LIN {X 0,Y 195.698,Z 597.397,A -85,B 0,C 180,E1 -23899.728,E2 -23899.728} C_VEL
LIN {X 0,Y 185.905,Z 599.961,A -85,B 0,C 180,E1 -23902.781,E2 -23902.781} C_VEL
LIN {X 0,Y 177.033,Z 601.325,A -85,B 0,C 180,E1 -23906.236,E2 -23906.236} C_VEL
LIN {X 0,Y 169.221,Z 601.554,A -85,B 0,C 180,E1 -23910.108,E2 -23910.108} C_VEL
LIN {X 0,Y 162.575,Z 600.655,A -85,B 0,C 180,E1 -23914.387,E2 -23914.387} C_VEL
LIN {X 0,Y 157.166,Z 598.615,A -85,B 0,C 180,E1 -23919.039,E2 -23919.039} C_VEL
LIN {X 0,Y 153.01,Z 595.413,A -85,B 0,C 180,E1 -23924.003,E2 -23924.003} C_VEL
LIN {X 0,Y 150.309,Z 590.963,A -85,B 0,C 180,E1 -23929.221,E2 -23929.221} C_VEL
LIN {X 0,Y 149.048,Z 585.18,A -85,B 0,C 180,E1 -23934.589,E2 -23934.589} C_VEL
LIN {X 0,Y 148.592,Z 577.647,A -85,B 0,C 180,E1 -23940.001,E2 -23940.001} C_VEL
LIN {X 0,Y 148.719,Z 570.72,A -85,B 0,C 180,E1 -23944.066,E2 -23944.066} C_VEL
LIN {X 0,Y 149.243,Z 562.31,A -85,B 0,C 180,E1 -23948.122,E2 -23948.122} C_VEL
LIN {X 0,Y 150.203,Z 552.102,A -85,B 0,C 180,E1 -23952.156,E2 -23952.156} C_VEL
LIN {X 0,Y 151.448,Z 540.799,A -85,B 0,C 180,E1 -23955.822,E2 -23955.822} C_VEL
LIN {X 0,Y 153.043,Z 528.174,A -85,B 0,C 180,E1 -23959.099,E2 -23959.099} C_VEL
LIN {X 0,Y 153.526,Z 523.721,A -85,B 0,C 180,E1 -23960.081,E2 -23960.081} C_VEL
LIN {X 0,Y 151.149,Z 510.343,A -85,B 0,C 180,E1 -23962.599,E2 -23962.599} C_VEL
LIN {X 0,Y 149.173,Z 497.903,A -85,B 0,C 180,E1 -23964.527,E2 -23964.527} C_VEL
LIN {X 0,Y 149.561,Z 497.851,A -85,B 0,C 180,E1 -23971.126,E2 -23971.126} C_VEL
LIN {X 0,Y 149.776,Z 497.824,A -85,B 0,C 180,E1 -23974.27,E2 -23974.27} C_VEL
LIN {X 0,Y 149.993,Z 497.8,A -85,B 0,C 180,E1 -23977.527,E2 -23977.527} C_VEL
LIN {X 0,Y 150.099,Z 497.782,A -85,B 0,C 180,E1 -23981.482,E2 -23981.482} C_VEL
LIN {X 0,Y 150.128,Z 497.783,A -85,B 0,C 180,E1 -23985.396,E2 -23985.396} C_VEL
LIN {X 0,Y 150.159,Z 497.776,A -85,B 0,C 180,E1 -23989.061,E2 -23989.061} C_VEL
LIN {X 0,Y 150.219,Z 497.772,A -85,B 0,C 180,E1 -23992.69,E2 -23992.69} C_VEL
LIN {X 0,Y 150.222,Z 497.77,A -85,B 0,C 180,E1 -23997.366,E2 -23997.366} C_VEL
LIN {X 0,Y 150.248,Z 497.769,A -85,B 0,C 180,E1 -24002.718,E2 -24002.718} C_VEL
LIN {X 0,Y 150.355,Z 497.751,A -85,B 0,C 180,E1 -24009.208,E2 -24009.208} C_VEL
LIN {X 0,Y 150.387,Z 497.752,A -85,B 0,C 180,E1 -24013.716,E2 -24013.716} C_VEL
LIN {X 0,Y 150.693,Z 497.711,A -85,B 0,C 180,E1 -24019.248,E2 -24019.248} C_VEL
LIN {X 0,Y 150.767,Z 497.706,A -85,B 0,C 180,E1 -24021.961,E2 -24021.961} C_VEL
LIN {X 0,Y 151.222,Z 497.65,A -85,B 0,C 180,E1 -24030,E2 -24030} C_VEL
LIN {X 0,Y 150.706,Z 497.714,A -85,B 0,C 180,E1 -24038.042,E2 -24038.042} C_VEL
LIN {X 0,Y 150.581,Z 497.726,A -85,B 0,C 180,E1 -24041.438,E2 -24041.438} C_VEL
LIN {X 0,Y 150.366,Z 497.755,A -85,B 0,C 180,E1 -24046.286,E2 -24046.286} C_VEL
LIN {X 0,Y 150.355,Z 497.751,A -85,B 0,C 180,E1 -24050.792,E2 -24050.792} C_VEL
LIN {X 0,Y 150.248,Z 497.769,A -85,B 0,C 180,E1 -24057.282,E2 -24057.282} C_VEL
LIN {X 0,Y 150.222,Z 497.77,A -85,B 0,C 180,E1 -24062.634,E2 -24062.634} C_VEL
LIN {X 0,Y 150.214,Z 497.773,A -85,B 0,C 180,E1 -24067.461,E2 -24067.461} C_VEL
LIN {X 0,Y 150.156,Z 497.778,A -85,B 0,C 180,E1 -24071.506,E2 -24071.506} C_VEL
LIN {X 0,Y 150.129,Z 497.784,A -85,B 0,C 180,E1 -24075.395,E2 -24075.395} C_VEL
LIN {X 0,Y 150.131,Z 497.778,A -85,B 0,C 180,E1 -24079.051,E2 -24079.051} C_VEL
LIN {X 0,Y 150.078,Z 497.79,A -85,B 0,C 180,E1 -24082.759,E2 -24082.759} C_VEL
LIN {X 0,Y 149.751,Z 497.826,A -85,B 0,C 180,E1 -24087.647,E2 -24087.647} C_VEL
LIN {X 0,Y 149.178,Z 497.898,A -85,B 0,C 180,E1 -24094.912,E2 -24094.912} C_VEL
LIN {X 0,Y 149.136,Z 497.907,A -85,B 0,C 180,E1 -24096.018,E2 -24096.018} C_VEL
LIN {X 0,Y 151.509,Z 512.126,A -85,B 0,C 180,E1 -24098.216,E2 -24098.216} C_VEL
LIN {X 0,Y 153.423,Z 522.893,A -85,B 0,C 180,E1 -24100.254,E2 -24100.254} C_VEL
LIN {X 0,Y 151.972,Z 535.306,A -85,B 0,C 180,E1 -24103.199,E2 -24103.199} C_VEL
LIN {X 0,Y 150.644,Z 546.515,A -85,B 0,C 180,E1 -24106.51,E2 -24106.51} C_VEL
LIN {X 0,Y 149.6,Z 556.661,A -85,B 0,C 180,E1 -24110.159,E2 -24110.159} C_VEL
LIN {X 0,Y 148.959,Z 565.049,A -85,B 0,C 180,E1 -24113.76,E2 -24113.76} C_VEL
LIN {X 0,Y 148.687,Z 573.127,A -85,B 0,C 180,E1 -24117.968,E2 -24117.968} C_VEL
LIN {X 0,Y 148.708,Z 580.512,A -85,B 0,C 180,E1 -24122.708,E2 -24122.708} C_VEL
LIN {X 0,Y 149.245,Z 585.686,A -85,B 0,C 180,E1 -24126.76,E2 -24126.76} C_VEL
LIN {X 0,Y 150.765,Z 591.202,A -85,B 0,C 180,E1 -24132.108,E2 -24132.108} C_VEL
LIN {X 0,Y 152.915,Z 594.451,A -85,B 0,C 180,E1 -24136.007,E2 -24136.007} C_VEL
LIN {X 0,Y 156.871,Z 597.69,A -85,B 0,C 180,E1 -24141.002,E2 -24141.002} C_VEL
LIN {X 0,Y 162.42,Z 599.76,A -85,B 0,C 180,E1 -24145.639,E2 -24145.639} C_VEL
LIN {X 0,Y 168.979,Z 600.68,A -85,B 0,C 180,E1 -24149.939,E2 -24149.939} C_VEL
LIN {X 0,Y 176.86,Z 600.442,A -85,B 0,C 180,E1 -24153.802,E2 -24153.802} C_VEL
LIN {X 0,Y 185.647,Z 599.082,A -85,B 0,C 180,E1 -24157.28,E2 -24157.28} C_VEL
LIN {X 0,Y 195.377,Z 596.535,A -85,B 0,C 180,E1 -24160.352,E2 -24160.352} C_VEL
LIN {X 0,Y 200.299,Z 594.929,A -85,B 0,C 180,E1 -24161.81,E2 -24161.81} C_VEL
LIN {X 0,Y 200.671,Z 594.93,A -85,B 0,C 180,E1 -24162.652,E2 -24162.652} C_VEL
LIN {X 0,Y 200.082,Z 595.451,A -85,B 0,C 180,E1 -24163.939,E2 -24163.939} C_VEL
LIN {X 0,Y 192.789,Z 598.957,A -85,B 0,C 180,E1 -24166.81,E2 -24166.81} C_VEL
LIN {X 0,Y 184.321,Z 602.303,A -85,B 0,C 180,E1 -24169.594,E2 -24169.594} C_VEL
LIN {X 0,Y 175.329,Z 605.126,A -85,B 0,C 180,E1 -24173.039,E2 -24173.039} C_VEL
LIN {X 0,Y 167.437,Z 606.911,A -85,B 0,C 180,E1 -24176.93,E2 -24176.93} C_VEL
LIN {X 0,Y 160.914,Z 607.677,A -85,B 0,C 180,E1 -24181.286,E2 -24181.286} C_VEL
LIN {X 0,Y 155.792,Z 607.424,A -85,B 0,C 180,E1 -24186.046,E2 -24186.046} C_VEL
LIN {X 0,Y 151.961,Z 606.089,A -85,B 0,C 180,E1 -24191.111,E2 -24191.111} C_VEL
LIN {X 0,Y 149.995,Z 603.727,A -85,B 0,C 180,E1 -24196.451,E2 -24196.451} C_VEL
LIN {X 0,Y 149.516,Z 600.172,A -85,B 0,C 180,E1 -24201.893,E2 -24201.893} C_VEL
LIN {X 0,Y 150.323,Z 595.194,A -85,B 0,C 180,E1 -24207.32,E2 -24207.32} C_VEL
LIN {X 0,Y 150.968,Z 592.887,A -85,B 0,C 180,E1 -24209.417,E2 -24209.417} C_VEL
LIN {X 0,Y 150.235,Z 596.744,A -85,B 0,C 180,E1 -24212.681,E2 -24212.681} C_VEL
LIN {X 0,Y 149.476,Z 601.603,A -85,B 0,C 180,E1 -24218.109,E2 -24218.109} C_VEL
LIN {X 0,Y 149.995,Z 605.064,A -85,B 0,C 180,E1 -24223.549,E2 -24223.549} C_VEL
LIN {X 0,Y 151.974,Z 607.36,A -85,B 0,C 180,E1 -24228.888,E2 -24228.888} C_VEL
LIN {X 0,Y 155.742,Z 608.606,A -85,B 0,C 180,E1 -24233.962,E2 -24233.962} C_VEL
LIN {X 0,Y 160.842,Z 608.816,A -85,B 0,C 180,E1 -24238.728,E2 -24238.728} C_VEL
LIN {X 0,Y 167.323,Z 608.017,A -85,B 0,C 180,E1 -24243.095,E2 -24243.095} C_VEL
LIN {X 0,Y 175.233,Z 606.214,A -85,B 0,C 180,E1 -24246.985,E2 -24246.985} C_VEL
LIN {X 0,Y 184.257,Z 603.388,A -85,B 0,C 180,E1 -24250.423,E2 -24250.423} C_VEL
LIN {X 0,Y 192.551,Z 600.121,A -85,B 0,C 180,E1 -24253.115,E2 -24253.115} C_VEL
LIN {X 0,Y 193.601,Z 599.632,A -85,B 0,C 180,E1 -24253.603,E2 -24253.603} C_VEL
LIN {X 0,Y 194.551,Z 599.052,A -85,B 0,C 180,E1 -24254.504,E2 -24254.504} C_VEL
LIN {X 0,Y 194.188,Z 598.82,A -85,B 0,C 180,E1 -24255.686,E2 -24255.686} C_VEL
LIN {X 0,Y 193.049,Z 598.915,A -85,B 0,C 180,E1 -24256.645,E2 -24256.645} C_VEL
LIN {X 0,Y 189.995,Z 599.516,A -85,B 0,C 180,E1 -24258.205,E2 -24258.205} C_VEL
LIN {X 0,Y 186.113,Z 600.31,A -85,B 0,C 180,E1 -24259.607,E2 -24259.607} C_VEL
LIN {X 0,Y 175.487,Z 601.989,A -85,B 0,C 180,E1 -24263.223,E2 -24263.223} C_VEL
LIN {X 0,Y 167.088,Z 602.317,A -85,B 0,C 180,E1 -24266.853,E2 -24266.853} C_VEL
LIN {X 0,Y 159.474,Z 601.564,A -85,B 0,C 180,E1 -24271.003,E2 -24271.003} C_VEL
LIN {X 0,Y 153.166,Z 599.679,A -85,B 0,C 180,E1 -24275.609,E2 -24275.609} C_VEL
LIN {X 0,Y 148.269,Z 596.683,A -85,B 0,C 180,E1 -24280.622,E2 -24280.622} C_VEL
LIN {X 0,Y 144.606,Z 592.483,A -85,B 0,C 180,E1 -24285.937,E2 -24285.937} C_VEL
LIN {X 0,Y 142.655,Z 587.019,A -85,B 0,C 180,E1 -24291.501,E2 -24291.501} C_VEL
LIN {X 0,Y 141.933,Z 581.951,A -85,B 0,C 180,E1 -24295.741,E2 -24295.741} C_VEL
LIN {X 0,Y 141.696,Z 574.718,A -85,B 0,C 180,E1 -24300.711,E2 -24300.711} C_VEL
LIN {X 0,Y 141.959,Z 565.75,A -85,B 0,C 180,E1 -24305.683,E2 -24305.683} C_VEL
LIN {X 0,Y 142.577,Z 557.063,A -85,B 0,C 180,E1 -24309.647,E2 -24309.647} C_VEL
LIN {X 0,Y 143.592,Z 546.908,A -85,B 0,C 180,E1 -24313.444,E2 -24313.444} C_VEL
LIN {X 0,Y 144.929,Z 535.658,A -85,B 0,C 180,E1 -24316.916,E2 -24316.916} C_VEL
LIN {X 0,Y 146.287,Z 524.84,A -85,B 0,C 180,E1 -24319.652,E2 -24319.652} C_VEL
LIN {X 0,Y 146.362,Z 523.284,A -85,B 0,C 180,E1 -24320,E2 -24320} C_VEL
LIN {X 0,Y 144.073,Z 510.803,A -85,B 0,C 180,E1 -24322.438,E2 -24322.438} C_VEL
LIN {X 0,Y 142.135,Z 498.779,A -85,B 0,C 180,E1 -24324.367,E2 -24324.367} C_VEL
LIN {X 0,Y 142.325,Z 498.755,A -85,B 0,C 180,E1 -24329.591,E2 -24329.591} C_VEL
LIN {X 0,Y 142.66,Z 498.708,A -85,B 0,C 180,E1 -24333.124,E2 -24333.124} C_VEL
LIN {X 0,Y 142.929,Z 498.682,A -85,B 0,C 180,E1 -24338.118,E2 -24338.118} C_VEL
LIN {X 0,Y 143.025,Z 498.665,A -85,B 0,C 180,E1 -24343.468,E2 -24343.468} C_VEL
LIN {X 0,Y 143.07,Z 498.662,A -85,B 0,C 180,E1 -24347.465,E2 -24347.465} C_VEL
LIN {X 0,Y 143.109,Z 498.654,A -85,B 0,C 180,E1 -24351.792,E2 -24351.792} C_VEL
LIN {X 0,Y 143.189,Z 498.646,A -85,B 0,C 180,E1 -24357.323,E2 -24357.323} C_VEL
LIN {X 0,Y 143.194,Z 498.647,A -85,B 0,C 180,E1 -24362.063,E2 -24362.063} C_VEL
LIN {X 0,Y 143.28,Z 498.633,A -85,B 0,C 180,E1 -24368.746,E2 -24368.746} C_VEL
LIN {X 0,Y 143.321,Z 498.631,A -85,B 0,C 180,E1 -24372.889,E2 -24372.889} C_VEL
LIN {X 0,Y 143.607,Z 498.594,A -85,B 0,C 180,E1 -24378.711,E2 -24378.711} C_VEL
LIN {X 0,Y 143.689,Z 498.586,A -85,B 0,C 180,E1 -24381.562,E2 -24381.562} C_VEL
LIN {X 0,Y 144.18,Z 498.527,A -85,B 0,C 180,E1 -24390,E2 -24390} C_VEL
LIN {X 0,Y 143.628,Z 498.594,A -85,B 0,C 180,E1 -24398.441,E2 -24398.441} C_VEL
LIN {X 0,Y 143.509,Z 498.606,A -85,B 0,C 180,E1 -24401.63,E2 -24401.63} C_VEL
LIN {X 0,Y 143.306,Z 498.633,A -85,B 0,C 180,E1 -24407.113,E2 -24407.113} C_VEL
LIN {X 0,Y 143.28,Z 498.633,A -85,B 0,C 180,E1 -24411.254,E2 -24411.254} C_VEL
LIN {X 0,Y 143.194,Z 498.647,A -85,B 0,C 180,E1 -24417.937,E2 -24417.937} C_VEL
LIN {X 0,Y 143.172,Z 498.649,A -85,B 0,C 180,E1 -24423.435,E2 -24423.435} C_VEL
LIN {X 0,Y 143.078,Z 498.657,A -85,B 0,C 180,E1 -24429.685,E2 -24429.685} C_VEL
LIN {X 0,Y 143.059,Z 498.665,A -85,B 0,C 180,E1 -24433.454,E2 -24433.454} C_VEL
LIN {X 0,Y 143.04,Z 498.663,A -85,B 0,C 180,E1 -24437.476,E2 -24437.476} C_VEL
LIN {X 0,Y 143.001,Z 498.673,A -85,B 0,C 180,E1 -24441.845,E2 -24441.845} C_VEL
LIN {X 0,Y 142.732,Z 498.699,A -85,B 0,C 180,E1 -24447.204,E2 -24447.204} C_VEL
LIN {X 0,Y 142.205,Z 498.77,A -85,B 0,C 180,E1 -24453.589,E2 -24453.589} C_VEL
LIN {X 0,Y 142.1,Z 498.779,A -85,B 0,C 180,E1 -24456.16,E2 -24456.16} C_VEL
LIN {X 0,Y 144.624,Z 513.6,A -85,B 0,C 180,E1 -24458.611,E2 -24458.611} C_VEL
LIN {X 0,Y 146.197,Z 522.332,A -85,B 0,C 180,E1 -24460.335,E2 -24460.335} C_VEL
LIN {X 0,Y 145.634,Z 528.278,A -85,B 0,C 180,E1 -24461.718,E2 -24461.718} C_VEL
LIN {X 0,Y 144.143,Z 540.798,A -85,B 0,C 180,E1 -24465.168,E2 -24465.168} C_VEL
LIN {X 0,Y 143.042,Z 551.16,A -85,B 0,C 180,E1 -24468.665,E2 -24468.665} C_VEL
LIN {X 0,Y 142.204,Z 561.169,A -85,B 0,C 180,E1 -24472.825,E2 -24472.825} C_VEL
LIN {X 0,Y 141.753,Z 571.068,A -85,B 0,C 180,E1 -24477.868,E2 -24477.868} C_VEL
LIN {X 0,Y 141.731,Z 577.84,A -85,B 0,C 180,E1 -24482.131,E2 -24482.131} C_VEL
LIN {X 0,Y 142.324,Z 584.32,A -85,B 0,C 180,E1 -24487.091,E2 -24487.091} C_VEL
LIN {X 0,Y 143.927,Z 590.206,A -85,B 0,C 180,E1 -24492.693,E2 -24492.693} C_VEL
LIN {X 0,Y 146.148,Z 593.742,A -85,B 0,C 180,E1 -24496.769,E2 -24496.769} C_VEL
LIN {X 0,Y 150.296,Z 597.35,A -85,B 0,C 180,E1 -24501.967,E2 -24501.967} C_VEL
LIN {X 0,Y 156.063,Z 599.826,A -85,B 0,C 180,E1 -24506.764,E2 -24506.764} C_VEL
LIN {X 0,Y 162.897,Z 601.174,A -85,B 0,C 180,E1 -24511.179,E2 -24511.179} C_VEL
LIN {X 0,Y 171.052,Z 601.383,A -85,B 0,C 180,E1 -24515.114,E2 -24515.114} C_VEL
LIN {X 0,Y 180.143,Z 600.481,A -85,B 0,C 180,E1 -24518.624,E2 -24518.624} C_VEL
LIN {X 0,Y 192.327,Z 597.879,A -85,B 0,C 180,E1 -24522.318,E2 -24522.318} C_VEL
LIN {X 0,Y 193.424,Z 597.599,A -85,B 0,C 180,E1 -24522.62,E2 -24522.62} C_VEL
LIN {X 0,Y 193.141,Z 597.833,A -85,B 0,C 180,E1 -24523.301,E2 -24523.301} C_VEL
LIN {X 0,Y 187.979,Z 599.933,A -85,B 0,C 180,E1 -24525.264,E2 -24525.264} C_VEL
LIN {X 0,Y 178.992,Z 602.901,A -85,B 0,C 180,E1 -24528.126,E2 -24528.126} C_VEL
LIN {X 0,Y 169.716,Z 605.248,A -85,B 0,C 180,E1 -24531.599,E2 -24531.599} C_VEL
LIN {X 0,Y 161.541,Z 606.599,A -85,B 0,C 180,E1 -24535.557,E2 -24535.557} C_VEL
LIN {X 0,Y 154.751,Z 606.96,A -85,B 0,C 180,E1 -24540.029,E2 -24540.029} C_VEL
LIN {X 0,Y 149.379,Z 606.337,A -85,B 0,C 180,E1 -24544.948,E2 -24544.948} C_VEL
LIN {X 0,Y 145.387,Z 604.683,A -85,B 0,C 180,E1 -24550.222,E2 -24550.222} C_VEL
LIN {X 0,Y 143.292,Z 602.031,A -85,B 0,C 180,E1 -24555.804,E2 -24555.804} C_VEL
LIN {X 0,Y 142.768,Z 598.17,A -85,B 0,C 180,E1 -24561.507,E2 -24561.507} C_VEL
LIN {X 0,Y 143.268,Z 594.348,A -85,B 0,C 180,E1 -24565.78,E2 -24565.78} C_VEL
LIN {X 0,Y 144.265,Z 590.518,A -85,B 0,C 180,E1 -24569.477,E2 -24569.477} C_VEL
LIN {X 0,Y 143.521,Z 594.455,A -85,B 0,C 180,E1 -24572.807,E2 -24572.807} C_VEL
LIN {X 0,Y 142.718,Z 599.608,A -85,B 0,C 180,E1 -24578.496,E2 -24578.496} C_VEL
LIN {X 0,Y 143.292,Z 603.359,A -85,B 0,C 180,E1 -24584.196,E2 -24584.196} C_VEL
LIN {X 0,Y 145.395,Z 605.939,A -85,B 0,C 180,E1 -24589.777,E2 -24589.777} C_VEL
LIN {X 0,Y 149.329,Z 607.531,A -85,B 0,C 180,E1 -24595.061,E2 -24595.061} C_VEL
LIN {X 0,Y 154.681,Z 608.094,A -85,B 0,C 180,E1 -24599.986,E2 -24599.986} C_VEL
LIN {X 0,Y 161.445,Z 607.693,A -85,B 0,C 180,E1 -24604.466,E2 -24604.466} C_VEL
LIN {X 0,Y 169.631,Z 606.322,A -85,B 0,C 180,E1 -24608.423,E2 -24608.423} C_VEL
LIN {X 0,Y 178.93,Z 603.954,A -85,B 0,C 180,E1 -24611.892,E2 -24611.892} C_VEL
LIN {X 0,Y 183.94,Z 602.402,A -85,B 0,C 180,E1 -24613.452,E2 -24613.452} C_VEL
LIN {X 0,Y 188.35,Z 600.741,A -85,B 0,C 180,E1 -24615.15,E2 -24615.15} C_VEL
LIN {X 0,Y 190.841,Z 599.408,A -85,B 0,C 180,E1 -24617.437,E2 -24617.437} C_VEL
LIN {X 0,Y 190.33,Z 599.383,A -85,B 0,C 180,E1 -24618.345,E2 -24618.345} C_VEL
LIN {X 0,Y 186.113,Z 600.31,A -85,B 0,C 180,E1 -24619.607,E2 -24619.607} C_VEL
LIN {X 0,Y 181.594,Z 601.229,A -85,B 0,C 180,E1 -24620.761,E2 -24620.761} C_VEL
LIN {X 0,Y 173.127,Z 602.455,A -85,B 0,C 180,E1 -24622.382,E2 -24622.382} C_VEL
LIN {X 0,Y 164.881,Z 602.98,A -85,B 0,C 180,E1 -24624.204,E2 -24624.204} C_VEL
LIN {X 0,Y 160.794,Z 602.817,A -85,B 0,C 180,E1 -24625.684,E2 -24625.684} C_VEL
LIN {X 0,Y 153.323,Z 601.682,A -85,B 0,C 180,E1 -24629.721,E2 -24629.721} C_VEL
LIN {X 0,Y 146.748,Z 599.415,A -85,B 0,C 180,E1 -24634.468,E2 -24634.468} C_VEL
LIN {X 0,Y 141.636,Z 596.05,A -85,B 0,C 180,E1 -24639.676,E2 -24639.676} C_VEL
LIN {X 0,Y 137.825,Z 591.457,A -85,B 0,C 180,E1 -24645.229,E2 -24645.229} C_VEL
LIN {X 0,Y 135.778,Z 585.648,A -85,B 0,C 180,E1 -24651.067,E2 -24651.067} C_VEL
LIN {X 0,Y 134.956,Z 579.252,A -85,B 0,C 180,E1 -24656.268,E2 -24656.268} C_VEL
LIN {X 0,Y 134.824,Z 571.474,A -85,B 0,C 180,E1 -24661.494,E2 -24661.494} C_VEL
LIN {X 0,Y 135.21,Z 562.075,A -85,B 0,C 180,E1 -24666.525,E2 -24666.525} C_VEL
LIN {X 0,Y 136.074,Z 551.25,A -85,B 0,C 180,E1 -24671.243,E2 -24671.243} C_VEL
LIN {X 0,Y 137.297,Z 540.041,A -85,B 0,C 180,E1 -24675.21,E2 -24675.21} C_VEL
LIN {X 0,Y 138.87,Z 527.241,A -85,B 0,C 180,E1 -24678.823,E2 -24678.823} C_VEL
LIN {X 0,Y 139.213,Z 524.26,A -85,B 0,C 180,E1 -24679.54,E2 -24679.54} C_VEL
LIN {X 0,Y 137.782,Z 515.546,A -85,B 0,C 180,E1 -24681.399,E2 -24681.399} C_VEL
LIN {X 0,Y 135.334,Z 501.393,A -85,B 0,C 180,E1 -24683.925,E2 -24683.925} C_VEL
LIN {X 0,Y 135.094,Z 499.655,A -85,B 0,C 180,E1 -24684.282,E2 -24684.282} C_VEL
LIN {X 0,Y 135.393,Z 499.616,A -85,B 0,C 180,E1 -24691.272,E2 -24691.272} C_VEL
LIN {X 0,Y 135.68,Z 499.582,A -85,B 0,C 180,E1 -24694.736,E2 -24694.736} C_VEL
LIN {X 0,Y 135.926,Z 499.551,A -85,B 0,C 180,E1 -24699.143,E2 -24699.143} C_VEL
LIN {X 0,Y 135.972,Z 499.544,A -85,B 0,C 180,E1 -24703.646,E2 -24703.646} C_VEL
LIN {X 0,Y 136.034,Z 499.54,A -85,B 0,C 180,E1 -24707.807,E2 -24707.807} C_VEL
LIN {X 0,Y 136.058,Z 499.532,A -85,B 0,C 180,E1 -24711.694,E2 -24711.694} C_VEL
LIN {X 0,Y 136.093,Z 499.532,A -85,B 0,C 180,E1 -24715.718,E2 -24715.718} C_VEL
LIN {X 0,Y 136.15,Z 499.526,A -85,B 0,C 180,E1 -24722.317,E2 -24722.317} C_VEL
LIN {X 0,Y 136.247,Z 499.509,A -85,B 0,C 180,E1 -24728.833,E2 -24728.833} C_VEL
LIN {X 0,Y 136.29,Z 499.505,A -85,B 0,C 180,E1 -24735.058,E2 -24735.058} C_VEL
LIN {X 0,Y 136.505,Z 499.477,A -85,B 0,C 180,E1 -24738.115,E2 -24738.115} C_VEL
LIN {X 0,Y 136.613,Z 499.467,A -85,B 0,C 180,E1 -24741.122,E2 -24741.122} C_VEL
LIN {X 0,Y 137.137,Z 499.404,A -85,B 0,C 180,E1 -24750,E2 -24750} C_VEL
LIN {X 0,Y 136.554,Z 499.474,A -85,B 0,C 180,E1 -24758.882,E2 -24758.882} C_VEL
LIN {X 0,Y 136.444,Z 499.484,A -85,B 0,C 180,E1 -24761.89,E2 -24761.89} C_VEL
LIN {X 0,Y 136.246,Z 499.514,A -85,B 0,C 180,E1 -24768.029,E2 -24768.029} C_VEL
LIN {X 0,Y 136.202,Z 499.513,A -85,B 0,C 180,E1 -24771.749,E2 -24771.749} C_VEL
LIN {X 0,Y 136.104,Z 499.528,A -85,B 0,C 180,E1 -24778.616,E2 -24778.616} C_VEL
LIN {X 0,Y 136.082,Z 499.533,A -85,B 0,C 180,E1 -24784.618,E2 -24784.618} C_VEL
LIN {X 0,Y 136.053,Z 499.532,A -85,B 0,C 180,E1 -24789.208,E2 -24789.208} C_VEL
LIN {X 0,Y 136,Z 499.545,A -85,B 0,C 180,E1 -24793.657,E2 -24793.657} C_VEL
LIN {X 0,Y 135.982,Z 499.54,A -85,B 0,C 180,E1 -24797.786,E2 -24797.786} C_VEL
LIN {X 0,Y 135.953,Z 499.55,A -85,B 0,C 180,E1 -24801.659,E2 -24801.659} C_VEL
LIN {X 0,Y 135.745,Z 499.57,A -85,B 0,C 180,E1 -24805.933,E2 -24805.933} C_VEL
LIN {X 0,Y 135.223,Z 499.64,A -85,B 0,C 180,E1 -24812.11,E2 -24812.11} C_VEL
LIN {X 0,Y 135.096,Z 499.651,A -85,B 0,C 180,E1 -24816.378,E2 -24816.378} C_VEL
LIN {X 0,Y 137.396,Z 513.137,A -85,B 0,C 180,E1 -24818.693,E2 -24818.693} C_VEL
LIN {X 0,Y 139.149,Z 523.438,A -85,B 0,C 180,E1 -24820.834,E2 -24820.834} C_VEL
LIN {X 0,Y 137.474,Z 536.858,A -85,B 0,C 180,E1 -24824.431,E2 -24824.431} C_VEL
LIN {X 0,Y 136.343,Z 547.769,A -85,B 0,C 180,E1 -24828.1,E2 -24828.1} C_VEL
LIN {X 0,Y 135.307,Z 559.508,A -85,B 0,C 180,E1 -24832.96,E2 -24832.96} C_VEL
LIN {X 0,Y 134.855,Z 568.8,A -85,B 0,C 180,E1 -24837.759,E2 -24837.759} C_VEL
LIN {X 0,Y 134.868,Z 575.931,A -85,B 0,C 180,E1 -24842.239,E2 -24842.239} C_VEL
LIN {X 0,Y 135.456,Z 582.799,A -85,B 0,C 180,E1 -24847.452,E2 -24847.452} C_VEL
LIN {X 0,Y 137.113,Z 589.071,A -85,B 0,C 180,E1 -24853.334,E2 -24853.334} C_VEL
LIN {X 0,Y 140.397,Z 593.967,A -85,B 0,C 180,E1 -24858.988,E2 -24858.988} C_VEL
LIN {X 0,Y 143.774,Z 596.869,A -85,B 0,C 180,E1 -24863.02,E2 -24863.02} C_VEL
LIN {X 0,Y 149.763,Z 599.734,A -85,B 0,C 180,E1 -24867.987,E2 -24867.987} C_VEL
LIN {X 0,Y 156.883,Z 601.486,A -85,B 0,C 180,E1 -24872.518,E2 -24872.518} C_VEL
LIN {X 0,Y 165.34,Z 602.132,A -85,B 0,C 180,E1 -24876.518,E2 -24876.518} C_VEL
LIN {X 0,Y 174.715,Z 601.69,A -85,B 0,C 180,E1 -24880.061,E2 -24880.061} C_VEL
LIN {X 0,Y 179.761,Z 601.068,A -85,B 0,C 180,E1 -24881.654,E2 -24881.654} C_VEL
LIN {X 0,Y 183.862,Z 600.524,A -85,B 0,C 180,E1 -24883.426,E2 -24883.426} C_VEL
LIN {X 0,Y 178.903,Z 602.017,A -85,B 0,C 180,E1 -24885,E2 -24885} C_VEL
LIN {X 0,Y 168.885,Z 604.384,A -85,B 0,C 180,E1 -24888.254,E2 -24888.254} C_VEL
LIN {X 0,Y 159.927,Z 605.788,A -85,B 0,C 180,E1 -24892.031,E2 -24892.031} C_VEL
LIN {X 0,Y 151.774,Z 606.22,A -85,B 0,C 180,E1 -24896.46,E2 -24896.46} C_VEL
LIN {X 0,Y 145.667,Z 605.717,A -85,B 0,C 180,E1 -24901.153,E2 -24901.153} C_VEL
LIN {X 0,Y 140.776,Z 604.247,A -85,B 0,C 180,E1 -24906.46,E2 -24906.46} C_VEL
LIN {X 0,Y 137.516,Z 601.771,A -85,B 0,C 180,E1 -24912.143,E2 -24912.143} C_VEL
LIN {X 0,Y 136.069,Z 597.67,A -85,B 0,C 180,E1 -24918.916,E2 -24918.916} C_VEL
LIN {X 0,Y 136.36,Z 593.416,A -85,B 0,C 180,E1 -24924.083,E2 -24924.083} C_VEL
LIN {X 0,Y 137.676,Z 587.892,A -85,B 0,C 180,E1 -24929.452,E2 -24929.452} C_VEL
LIN {X 0,Y 136.52,Z 593.578,A -85,B 0,C 180,E1 -24934.429,E2 -24934.429} C_VEL
LIN {X 0,Y 136.057,Z 599.045,A -85,B 0,C 180,E1 -24941.057,E2 -24941.057} C_VEL
LIN {X 0,Y 136.63,Z 601.524,A -85,B 0,C 180,E1 -24944.903,E2 -24944.903} C_VEL
LIN {X 0,Y 138.871,Z 604.406,A -85,B 0,C 180,E1 -24950.748,E2 -24950.748} C_VEL
LIN {X 0,Y 143.001,Z 606.304,A -85,B 0,C 180,E1 -24956.252,E2 -24956.252} C_VEL
LIN {X 0,Y 148.6,Z 607.22,A -85,B 0,C 180,E1 -24961.349,E2 -24961.349} C_VEL
LIN {X 0,Y 155.662,Z 607.204,A -85,B 0,C 180,E1 -24965.94,E2 -24965.94} C_VEL
LIN {X 0,Y 164.134,Z 606.261,A -85,B 0,C 180,E1 -24969.962,E2 -24969.962} C_VEL
LIN {X 0,Y 173.716,Z 604.359,A -85,B 0,C 180,E1 -24973.454,E2 -24973.454} C_VEL
LIN {X 0,Y 178.874,Z 603.043,A -85,B 0,C 180,E1 -24975.01,E2 -24975.01} C_VEL
LIN {X 0,Y 182.905,Z 601.689,A -85,B 0,C 180,E1 -24976.892,E2 -24976.892} C_VEL
LIN {X 0,Y 180.033,Z 601.984,A -85,B 0,C 180,E1 -24978.423,E2 -24978.423} C_VEL
LIN {X 0,Y 169.91,Z 602.975,A -85,B 0,C 180,E1 -24981.804,E2 -24981.804} C_VEL
LIN {X 0,Y 160.794,Z 602.817,A -85,B 0,C 180,E1 -24985.684,E2 -24985.684} C_VEL
LIN {X 0,Y 156.842,Z 602.474,A -85,B 0,C 180,E1 -24987.265,E2 -24987.265} C_VEL
LIN {X 0,Y 149.307,Z 601.394,A -85,B 0,C 180,E1 -24989.651,E2 -24989.651} C_VEL
LIN {X 0,Y 142.286,Z 599.63,A -85,B 0,C 180,E1 -24992.298,E2 -24992.298} C_VEL
LIN {X 0,Y 139.235,Z 598.255,A -85,B 0,C 180,E1 -24994.272,E2 -24994.272} C_VEL
LIN {X 0,Y 133.927,Z 594.067,A -85,B 0,C 180,E1 -25000.057,E2 -25000.057} C_VEL
LIN {X 0,Y 130.313,Z 588.669,A -85,B 0,C 180,E1 -25006.113,E2 -25006.113} C_VEL
LIN {X 0,Y 128.66,Z 582.293,A -85,B 0,C 180,E1 -25012.152,E2 -25012.152} C_VEL
LIN {X 0,Y 127.98,Z 575.153,A -85,B 0,C 180,E1 -25017.64,E2 -25017.64} C_VEL
LIN {X 0,Y 127.98,Z 567.755,A -85,B 0,C 180,E1 -25022.361,E2 -25022.361} C_VEL
LIN {X 0,Y 128.385,Z 559.158,A -85,B 0,C 180,E1 -25026.933,E2 -25026.933} C_VEL
LIN {X 0,Y 129.252,Z 548.723,A -85,B 0,C 180,E1 -25031.452,E2 -25031.452} C_VEL
LIN {X 0,Y 130.532,Z 537.016,A -85,B 0,C 180,E1 -25035.618,E2 -25035.618} C_VEL
LIN {X 0,Y 132.104,Z 523.595,A -85,B 0,C 180,E1 -25039.422,E2 -25039.422} C_VEL
LIN {X 0,Y 129.838,Z 511.037,A -85,B 0,C 180,E1 -25042.101,E2 -25042.101} C_VEL
LIN {X 0,Y 128.082,Z 500.528,A -85,B 0,C 180,E1 -25043.977,E2 -25043.977} C_VEL
LIN {X 0,Y 128.178,Z 500.518,A -85,B 0,C 180,E1 -25049.57,E2 -25049.57} C_VEL
LIN {X 0,Y 128.633,Z 500.46,A -85,B 0,C 180,E1 -25054.96,E2 -25054.96} C_VEL
LIN {X 0,Y 128.854,Z 500.428,A -85,B 0,C 180,E1 -25060.884,E2 -25060.884} C_VEL
LIN {X 0,Y 128.918,Z 500.425,A -85,B 0,C 180,E1 -25065.131,E2 -25065.131} C_VEL
LIN {X 0,Y 128.96,Z 500.416,A -85,B 0,C 180,E1 -25069.728,E2 -25069.728} C_VEL
LIN {X 0,Y 128.995,Z 500.416,A -85,B 0,C 180,E1 -25074.811,E2 -25074.811} C_VEL
LIN {X 0,Y 129.036,Z 500.408,A -85,B 0,C 180,E1 -25080.647,E2 -25080.647} C_VEL
LIN {X 0,Y 129.112,Z 500.396,A -85,B 0,C 180,E1 -25087.602,E2 -25087.602} C_VEL
LIN {X 0,Y 129.164,Z 500.394,A -85,B 0,C 180,E1 -25090.945,E2 -25090.945} C_VEL
LIN {X 0,Y 129.422,Z 500.357,A -85,B 0,C 180,E1 -25097.815,E2 -25097.815} C_VEL
LIN {X 0,Y 129.535,Z 500.349,A -85,B 0,C 180,E1 -25100.632,E2 -25100.632} C_VEL
LIN {X 0,Y 130.092,Z 500.281,A -85,B 0,C 180,E1 -25110,E2 -25110} C_VEL
LIN {X 0,Y 129.479,Z 500.356,A -85,B 0,C 180,E1 -25119.372,E2 -25119.372} C_VEL
LIN {X 0,Y 129.348,Z 500.366,A -85,B 0,C 180,E1 -25122.553,E2 -25122.553} C_VEL
LIN {X 0,Y 129.157,Z 500.395,A -85,B 0,C 180,E1 -25129.056,E2 -25129.056} C_VEL
LIN {X 0,Y 129.112,Z 500.396,A -85,B 0,C 180,E1 -25132.398,E2 -25132.398} C_VEL
LIN {X 0,Y 129.039,Z 500.408,A -85,B 0,C 180,E1 -25139.373,E2 -25139.373} C_VEL
LIN {X 0,Y 128.995,Z 500.416,A -85,B 0,C 180,E1 -25145.189,E2 -25145.189} C_VEL
LIN {X 0,Y 128.953,Z 500.417,A -85,B 0,C 180,E1 -25150.845,E2 -25150.845} C_VEL
LIN {X 0,Y 128.918,Z 500.426,A -85,B 0,C 180,E1 -25155.129,E2 -25155.129} C_VEL
LIN {X 0,Y 128.913,Z 500.423,A -85,B 0,C 180,E1 -25159.751,E2 -25159.751} C_VEL
LIN {X 0,Y 128.724,Z 500.448,A -85,B 0,C 180,E1 -25164.982,E2 -25164.982} C_VEL
LIN {X 0,Y 128.209,Z 500.515,A -85,B 0,C 180,E1 -25171.291,E2 -25171.291} C_VEL
LIN {X 0,Y 128.093,Z 500.523,A -85,B 0,C 180,E1 -25176.667,E2 -25176.667} C_VEL
LIN {X 0,Y 130.603,Z 514.984,A -85,B 0,C 180,E1 -25179.32,E2 -25179.32} C_VEL
LIN {X 0,Y 132.009,Z 522.552,A -85,B 0,C 180,E1 -25180.968,E2 -25180.968} C_VEL
LIN {X 0,Y 130.608,Z 534.901,A -85,B 0,C 180,E1 -25184.391,E2 -25184.391} C_VEL
LIN {X 0,Y 129.449,Z 545.981,A -85,B 0,C 180,E1 -25188.173,E2 -25188.173} C_VEL
LIN {X 0,Y 128.512,Z 555.94,A -85,B 0,C 180,E1 -25192.316,E2 -25192.316} C_VEL
LIN {X 0,Y 128.041,Z 564.895,A -85,B 0,C 180,E1 -25196.853,E2 -25196.853} C_VEL
LIN {X 0,Y 127.986,Z 572.703,A -85,B 0,C 180,E1 -25201.573,E2 -25201.573} C_VEL
LIN {X 0,Y 128.396,Z 579.15,A -85,B 0,C 180,E1 -25206.284,E2 -25206.284} C_VEL
LIN {X 0,Y 129.716,Z 586.178,A -85,B 0,C 180,E1 -25212.516,E2 -25212.516} C_VEL
LIN {X 0,Y 132.761,Z 591.811,A -85,B 0,C 180,E1 -25218.519,E2 -25218.519} C_VEL
LIN {X 0,Y 137.309,Z 596.179,A -85,B 0,C 180,E1 -25224.171,E2 -25224.171} C_VEL
LIN {X 0,Y 143.546,Z 599.432,A -85,B 0,C 180,E1 -25229.314,E2 -25229.314} C_VEL
LIN {X 0,Y 150.953,Z 601.597,A -85,B 0,C 180,E1 -25233.965,E2 -25233.965} C_VEL
LIN {X 0,Y 159.717,Z 602.693,A -85,B 0,C 180,E1 -25238.027,E2 -25238.027} C_VEL
LIN {X 0,Y 169.389,Z 602.731,A -85,B 0,C 180,E1 -25241.593,E2 -25241.593} C_VEL
LIN {X 0,Y 173.964,Z 602.484,A -85,B 0,C 180,E1 -25243.349,E2 -25243.349} C_VEL
LIN {X 0,Y 163.669,Z 604.382,A -85,B 0,C 180,E1 -25246.603,E2 -25246.603} C_VEL
LIN {X 0,Y 154.41,Z 605.345,A -85,B 0,C 180,E1 -25250.415,E2 -25250.415} C_VEL
LIN {X 0,Y 145.768,Z 605.342,A -85,B 0,C 180,E1 -25255.047,E2 -25255.047} C_VEL
LIN {X 0,Y 139.576,Z 604.513,A -85,B 0,C 180,E1 -25259.766,E2 -25259.766} C_VEL
LIN {X 0,Y 134.449,Z 602.725,A -85,B 0,C 180,E1 -25265.28,E2 -25265.28} C_VEL
LIN {X 0,Y 131.009,Z 599.91,A -85,B 0,C 180,E1 -25271.224,E2 -25271.224} C_VEL
LIN {X 0,Y 129.542,Z 595.996,A -85,B 0,C 180,E1 -25277.564,E2 -25277.564} C_VEL
LIN {X 0,Y 129.748,Z 590.952,A -85,B 0,C 180,E1 -25283.781,E2 -25283.781} C_VEL
LIN {X 0,Y 131.156,Z 585.118,A -85,B 0,C 180,E1 -25289.424,E2 -25289.424} C_VEL
LIN {X 0,Y 130.262,Z 589.433,A -85,B 0,C 180,E1 -25293.093,E2 -25293.093} C_VEL
LIN {X 0,Y 129.383,Z 595.19,A -85,B 0,C 180,E1 -25299.379,E2 -25299.379} C_VEL
LIN {X 0,Y 130.032,Z 599.519,A -85,B 0,C 180,E1 -25305.679,E2 -25305.679} C_VEL
LIN {X 0,Y 132.44,Z 602.726,A -85,B 0,C 180,E1 -25311.806,E2 -25311.806} C_VEL
LIN {X 0,Y 136.764,Z 604.943,A -85,B 0,C 180,E1 -25317.548,E2 -25317.548} C_VEL
LIN {X 0,Y 144.863,Z 606.402,A -85,B 0,C 180,E1 -25324.438,E2 -25324.438} C_VEL
LIN {X 0,Y 154.246,Z 606.397,A -85,B 0,C 180,E1 -25329.635,E2 -25329.635} C_VEL
LIN {X 0,Y 163.566,Z 605.41,A -85,B 0,C 180,E1 -25333.431,E2 -25333.431} C_VEL
LIN {X 0,Y 173.854,Z 603.495,A -85,B 0,C 180,E1 -25336.69,E2 -25336.69} C_VEL
LIN {X 0,Y 169.652,Z 603.668,A -85,B 0,C 180,E1 -25338.485,E2 -25338.485} C_VEL
LIN {X 0,Y 159.904,Z 603.64,A -85,B 0,C 180,E1 -25342.026,E2 -25342.026} C_VEL
LIN {X 0,Y 151.167,Z 602.556,A -85,B 0,C 180,E1 -25346.09,E2 -25346.09} C_VEL
LIN {X 0,Y 143.712,Z 600.412,A -85,B 0,C 180,E1 -25350.723,E2 -25350.723} C_VEL
LIN {X 0,Y 139.235,Z 598.255,A -85,B 0,C 180,E1 -25354.272,E2 -25354.272} C_VEL
LIN {X 0,Y 136.414,Z 596.765,A -85,B 0,C 180,E1 -25356.328,E2 -25356.328} C_VEL
LIN {X 0,Y 130.631,Z 593.548,A -85,B 0,C 180,E1 -25359.503,E2 -25359.503} C_VEL
LIN {X 0,Y 125.438,Z 589.728,A -85,B 0,C 180,E1 -25362.894,E2 -25362.894} C_VEL
LIN {X 0,Y 123.641,Z 587.288,A -85,B 0,C 180,E1 -25365.236,E2 -25365.236} C_VEL
LIN {X 0,Y 121.873,Z 580.389,A -85,B 0,C 180,E1 -25371.712,E2 -25371.712} C_VEL
LIN {X 0,Y 121.151,Z 572.921,A -85,B 0,C 180,E1 -25377.507,E2 -25377.507} C_VEL
LIN {X 0,Y 121.177,Z 565.071,A -85,B 0,C 180,E1 -25382.494,E2 -25382.494} C_VEL
LIN {X 0,Y 121.603,Z 555.666,A -85,B 0,C 180,E1 -25387.473,E2 -25387.473} C_VEL
LIN {X 0,Y 122.451,Z 545.942,A -85,B 0,C 180,E1 -25391.735,E2 -25391.735} C_VEL
LIN {X 0,Y 123.823,Z 533.738,A -85,B 0,C 180,E1 -25396.064,E2 -25396.064} C_VEL
LIN {X 0,Y 124.995,Z 524.134,A -85,B 0,C 180,E1 -25398.864,E2 -25398.864} C_VEL
LIN {X 0,Y 123.373,Z 514.802,A -85,B 0,C 180,E1 -25401.022,E2 -25401.022} C_VEL
LIN {X 0,Y 121.076,Z 501.401,A -85,B 0,C 180,E1 -25403.69,E2 -25403.69} C_VEL
LIN {X 0,Y 121.225,Z 501.381,A -85,B 0,C 180,E1 -25411.452,E2 -25411.452} C_VEL
LIN {X 0,Y 121.62,Z 501.334,A -85,B 0,C 180,E1 -25416,E2 -25416} C_VEL
LIN {X 0,Y 121.795,Z 501.307,A -85,B 0,C 180,E1 -25421.397,E2 -25421.397} C_VEL
LIN {X 0,Y 121.846,Z 501.308,A -85,B 0,C 180,E1 -25426.199,E2 -25426.199} C_VEL
LIN {X 0,Y 121.877,Z 501.297,A -85,B 0,C 180,E1 -25430.631,E2 -25430.631} C_VEL
LIN {X 0,Y 121.948,Z 501.294,A -85,B 0,C 180,E1 -25434.808,E2 -25434.808} C_VEL
LIN {X 0,Y 121.945,Z 501.287,A -85,B 0,C 180,E1 -25439.827,E2 -25439.827} C_VEL
LIN {X 0,Y 121.987,Z 501.286,A -85,B 0,C 180,E1 -25446.216,E2 -25446.216} C_VEL
LIN {X 0,Y 122.053,Z 501.277,A -85,B 0,C 180,E1 -25449.788,E2 -25449.788} C_VEL
LIN {X 0,Y 122.268,Z 501.247,A -85,B 0,C 180,E1 -25456.708,E2 -25456.708} C_VEL
LIN {X 0,Y 122.461,Z 501.231,A -85,B 0,C 180,E1 -25460.086,E2 -25460.086} C_VEL
LIN {X 0,Y 122.614,Z 501.207,A -85,B 0,C 180,E1 -25466.714,E2 -25466.714} C_VEL
LIN {X 0,Y 123.045,Z 501.159,A -85,B 0,C 180,E1 -25470,E2 -25470} C_VEL
LIN {X 0,Y 122.426,Z 501.233,A -85,B 0,C 180,E1 -25476.593,E2 -25476.593} C_VEL
LIN {X 0,Y 122.321,Z 501.241,A -85,B 0,C 180,E1 -25482.376,E2 -25482.376} C_VEL
LIN {X 0,Y 122.112,Z 501.273,A -85,B 0,C 180,E1 -25486.724,E2 -25486.724} C_VEL
LIN {X 0,Y 122.027,Z 501.279,A -85,B 0,C 180,E1 -25492.85,E2 -25492.85} C_VEL
LIN {X 0,Y 121.953,Z 501.294,A -85,B 0,C 180,E1 -25497.454,E2 -25497.454} C_VEL
LIN {X 0,Y 121.915,Z 501.291,A -85,B 0,C 180,E1 -25501.253,E2 -25501.253} C_VEL
LIN {X 0,Y 121.915,Z 501.298,A -85,B 0,C 180,E1 -25506.189,E2 -25506.189} C_VEL
LIN {X 0,Y 121.886,Z 501.299,A -85,B 0,C 180,E1 -25511.444,E2 -25511.444} C_VEL
LIN {X 0,Y 121.837,Z 501.301,A -85,B 0,C 180,E1 -25518.581,E2 -25518.581} C_VEL
LIN {X 0,Y 121.692,Z 501.324,A -85,B 0,C 180,E1 -25524.722,E2 -25524.722} C_VEL
LIN {X 0,Y 121.232,Z 501.383,A -85,B 0,C 180,E1 -25530.409,E2 -25530.409} C_VEL
LIN {X 0,Y 121.114,Z 501.452,A -85,B 0,C 180,E1 -25537.045,E2 -25537.045} C_VEL
LIN {X 0,Y 123.51,Z 515.008,A -85,B 0,C 180,E1 -25539.667,E2 -25539.667} C_VEL
LIN {X 0,Y 124.899,Z 523.156,A -85,B 0,C 180,E1 -25541.547,E2 -25541.547} C_VEL
LIN {X 0,Y 123.384,Z 535.853,A -85,B 0,C 180,E1 -25545.316,E2 -25545.316} C_VEL
LIN {X 0,Y 122.254,Z 547.1,A -85,B 0,C 180,E1 -25549.505,E2 -25549.505} C_VEL
LIN {X 0,Y 121.494,Z 557.39,A -85,B 0,C 180,E1 -25554.189,E2 -25554.189} C_VEL
LIN {X 0,Y 121.186,Z 566.424,A -85,B 0,C 180,E1 -25559.168,E2 -25559.168} C_VEL
LIN {X 0,Y 121.397,Z 574.993,A -85,B 0,C 180,E1 -25564.981,E2 -25564.981} C_VEL
LIN {X 0,Y 122.145,Z 581.052,A -85,B 0,C 180,E1 -25569.939,E2 -25569.939} C_VEL
LIN {X 0,Y 124.358,Z 587.721,A -85,B 0,C 180,E1 -25576.413,E2 -25576.413} C_VEL
LIN {X 0,Y 128.351,Z 593.06,A -85,B 0,C 180,E1 -25582.537,E2 -25582.537} C_VEL
LIN {X 0,Y 133.95,Z 597.245,A -85,B 0,C 180,E1 -25588.177,E2 -25588.177} C_VEL
LIN {X 0,Y 141.049,Z 600.358,A -85,B 0,C 180,E1 -25593.236,E2 -25593.236} C_VEL
LIN {X 0,Y 149.538,Z 602.418,A -85,B 0,C 180,E1 -25597.659,E2 -25597.659} C_VEL
LIN {X 0,Y 159.068,Z 603.446,A -85,B 0,C 180,E1 -25601.508,E2 -25601.508} C_VEL
LIN {X 0,Y 163.769,Z 603.583,A -85,B 0,C 180,E1 -25603.152,E2 -25603.152} C_VEL
LIN {X 0,Y 153.649,Z 604.557,A -85,B 0,C 180,E1 -25606.677,E2 -25606.677} C_VEL
LIN {X 0,Y 144.592,Z 604.634,A -85,B 0,C 180,E1 -25610.811,E2 -25610.811} C_VEL
LIN {X 0,Y 136.879,Z 603.847,A -85,B 0,C 180,E1 -25615.612,E2 -25615.612} C_VEL
LIN {X 0,Y 130.694,Z 602.192,A -85,B 0,C 180,E1 -25621.055,E2 -25621.055} C_VEL
LIN {X 0,Y 126.127,Z 599.582,A -85,B 0,C 180,E1 -25627.042,E2 -25627.042} C_VEL
LIN {X 0,Y 123.549,Z 595.968,A -85,B 0,C 180,E1 -25633.476,E2 -25633.476} C_VEL
LIN {X 0,Y 122.879,Z 591.21,A -85,B 0,C 180,E1 -25640.12,E2 -25640.12} C_VEL
LIN {X 0,Y 123.475,Z 586.762,A -85,B 0,C 180,E1 -25645.102,E2 -25645.102} C_VEL
LIN {X 0,Y 124.689,Z 582.145,A -85,B 0,C 180,E1 -25649.394,E2 -25649.394} C_VEL
LIN {X 0,Y 123.373,Z 588.324,A -85,B 0,C 180,E1 -25654.902,E2 -25654.902} C_VEL
LIN {X 0,Y 122.815,Z 592.737,A -85,B 0,C 180,E1 -25659.885,E2 -25659.885} C_VEL
LIN {X 0,Y 123.511,Z 597.358,A -85,B 0,C 180,E1 -25666.53,E2 -25666.53} C_VEL
LIN {X 0,Y 126.111,Z 600.852,A -85,B 0,C 180,E1 -25672.961,E2 -25672.961} C_VEL
LIN {X 0,Y 130.645,Z 603.401,A -85,B 0,C 180,E1 -25678.957,E2 -25678.957} C_VEL
LIN {X 0,Y 139.147,Z 605.303,A -85,B 0,C 180,E1 -25686.088,E2 -25686.088} C_VEL
LIN {X 0,Y 148.883,Z 605.761,A -85,B 0,C 180,E1 -25691.366,E2 -25691.366} C_VEL
LIN {X 0,Y 158.501,Z 605.197,A -85,B 0,C 180,E1 -25695.19,E2 -25695.19} C_VEL
LIN {X 0,Y 163.71,Z 604.581,A -85,B 0,C 180,E1 -25696.87,E2 -25696.87} C_VEL
LIN {X 0,Y 159.306,Z 604.417,A -85,B 0,C 180,E1 -25698.567,E2 -25698.567} C_VEL
LIN {X 0,Y 149.754,Z 603.407,A -85,B 0,C 180,E1 -25702.404,E2 -25702.404} C_VEL
LIN {X 0,Y 141.268,Z 601.366,A -85,B 0,C 180,E1 -25706.822,E2 -25706.822} C_VEL
LIN {X 0,Y 134.135,Z 598.291,A -85,B 0,C 180,E1 -25711.865,E2 -25711.865} C_VEL
LIN {X 0,Y 128.546,Z 594.175,A -85,B 0,C 180,E1 -25717.499,E2 -25717.499} C_VEL
LIN {X 0,Y 123.867,Z 587.814,A -85,B 0,C 180,E1 -25724.699,E2 -25724.699} C_VEL
LIN {X 0,Y 123.641,Z 587.288,A -85,B 0,C 180,E1 -25725.236,E2 -25725.236} C_VEL
LIN {X 0,Y 122.128,Z 584.698,A -85,B 0,C 180,E1 -25727.595,E2 -25727.595} C_VEL
LIN {X 0,Y 118.419,Z 579.623,A -85,B 0,C 180,E1 -25731.241,E2 -25731.241} C_VEL
LIN {X 0,Y 115.153,Z 573.915,A -85,B 0,C 180,E1 -25734.956,E2 -25734.956} C_VEL
LIN {X 0,Y 114.423,Z 570.4,A -85,B 0,C 180,E1 -25737.355,E2 -25737.355} C_VEL
LIN {X 0,Y 114.395,Z 562.196,A -85,B 0,C 180,E1 -25742.642,E2 -25742.642} C_VEL
LIN {X 0,Y 114.778,Z 553.972,A -85,B 0,C 180,E1 -25747.035,E2 -25747.035} C_VEL
LIN {X 0,Y 115.697,Z 543.017,A -85,B 0,C 180,E1 -25751.947,E2 -25751.947} C_VEL
LIN {X 0,Y 116.956,Z 531.4,A -85,B 0,C 180,E1 -25756.177,E2 -25756.177} C_VEL
LIN {X 0,Y 117.849,Z 522.999,A -85,B 0,C 180,E1 -25758.697,E2 -25758.697} C_VEL
LIN {X 0,Y 115.292,Z 509.205,A -85,B 0,C 180,E1 -25761.877,E2 -25761.877} C_VEL
LIN {X 0,Y 114.079,Z 502.273,A -85,B 0,C 180,E1 -25763.282,E2 -25763.282} C_VEL
LIN {X 0,Y 114.132,Z 502.266,A -85,B 0,C 180,E1 -25770.448,E2 -25770.448} C_VEL
LIN {X 0,Y 114.587,Z 502.211,A -85,B 0,C 180,E1 -25777.123,E2 -25777.123} C_VEL
LIN {X 0,Y 114.729,Z 502.188,A -85,B 0,C 180,E1 -25782.685,E2 -25782.685} C_VEL
LIN {X 0,Y 114.803,Z 502.184,A -85,B 0,C 180,E1 -25787.67,E2 -25787.67} C_VEL
LIN {X 0,Y 114.815,Z 502.182,A -85,B 0,C 180,E1 -25792.728,E2 -25792.728} C_VEL
LIN {X 0,Y 114.872,Z 502.168,A -85,B 0,C 180,E1 -25798.932,E2 -25798.932} C_VEL
LIN {X 0,Y 114.95,Z 502.161,A -85,B 0,C 180,E1 -25806.508,E2 -25806.508} C_VEL
LIN {X 0,Y 115.022,Z 502.158,A -85,B 0,C 180,E1 -25812.211,E2 -25812.211} C_VEL
LIN {X 0,Y 115.29,Z 502.116,A -85,B 0,C 180,E1 -25817.257,E2 -25817.257} C_VEL
LIN {X 0,Y 115.397,Z 502.108,A -85,B 0,C 180,E1 -25819.472,E2 -25819.472} C_VEL
LIN {X 0,Y 115.541,Z 502.087,A -85,B 0,C 180,E1 -25826.513,E2 -25826.513} C_VEL
LIN {X 0,Y 115.996,Z 502.037,A -85,B 0,C 180,E1 -25830,E2 -25830} C_VEL
LIN {X 0,Y 115.367,Z 502.112,A -85,B 0,C 180,E1 -25836.998,E2 -25836.998} C_VEL
LIN {X 0,Y 115.255,Z 502.121,A -85,B 0,C 180,E1 -25842.666,E2 -25842.666} C_VEL
LIN {X 0,Y 115.015,Z 502.159,A -85,B 0,C 180,E1 -25847.79,E2 -25847.79} C_VEL
LIN {X 0,Y 114.95,Z 502.161,A -85,B 0,C 180,E1 -25853.492,E2 -25853.492} C_VEL
LIN {X 0,Y 114.872,Z 502.168,A -85,B 0,C 180,E1 -25861.068,E2 -25861.068} C_VEL
LIN {X 0,Y 114.805,Z 502.18,A -85,B 0,C 180,E1 -25867.747,E2 -25867.747} C_VEL
LIN {X 0,Y 114.795,Z 502.184,A -85,B 0,C 180,E1 -25872.72,E2 -25872.72} C_VEL
LIN {X 0,Y 114.773,Z 502.182,A -85,B 0,C 180,E1 -25877.655,E2 -25877.655} C_VEL
LIN {X 0,Y 114.661,Z 502.202,A -85,B 0,C 180,E1 -25882.828,E2 -25882.828} C_VEL
LIN {X 0,Y 114.217,Z 502.255,A -85,B 0,C 180,E1 -25889.48,E2 -25889.48} C_VEL
LIN {X 0,Y 114.109,Z 502.269,A -85,B 0,C 180,E1 -25897.497,E2 -25897.497} C_VEL
LIN {X 0,Y 116.703,Z 516.436,A -85,B 0,C 180,E1 -25900.428,E2 -25900.428} C_VEL
LIN {X 0,Y 117.764,Z 521.89,A -85,B 0,C 180,E1 -25901.74,E2 -25901.74} C_VEL
LIN {X 0,Y 116.647,Z 532.794,A -85,B 0,C 180,E1 -25905.073,E2 -25905.073} C_VEL
LIN {X 0,Y 115.509,Z 544.55,A -85,B 0,C 180,E1 -25909.482,E2 -25909.482} C_VEL
LIN {X 0,Y 114.678,Z 555.805,A -85,B 0,C 180,E1 -25914.725,E2 -25914.725} C_VEL
LIN {X 0,Y 114.458,Z 565.014,A -85,B 0,C 180,E1 -25919.999,E2 -25919.999} C_VEL
LIN {X 0,Y 114.629,Z 572.667,A -85,B 0,C 180,E1 -25925.276,E2 -25925.276} C_VEL
LIN {X 0,Y 115.434,Z 579.008,A -85,B 0,C 180,E1 -25930.523,E2 -25930.523} C_VEL
LIN {X 0,Y 117.752,Z 586.053,A -85,B 0,C 180,E1 -25937.362,E2 -25937.362} C_VEL
LIN {X 0,Y 121.939,Z 591.8,A -85,B 0,C 180,E1 -25943.793,E2 -25943.793} C_VEL
LIN {X 0,Y 127.807,Z 596.356,A -85,B 0,C 180,E1 -25949.663,E2 -25949.663} C_VEL
LIN {X 0,Y 135.185,Z 599.858,A -85,B 0,C 180,E1 -25954.88,E2 -25954.88} C_VEL
LIN {X 0,Y 144,Z 602.357,A -85,B 0,C 180,E1 -25959.38,E2 -25959.38} C_VEL
LIN {X 0,Y 152.194,Z 603.68,A -85,B 0,C 180,E1 -25962.67,E2 -25962.67} C_VEL
LIN {X 0,Y 152.051,Z 603.863,A -85,B 0,C 180,E1 -25963.544,E2 -25963.544} C_VEL
LIN {X 0,Y 139.217,Z 603.611,A -85,B 0,C 180,E1 -25968.984,E2 -25968.984} C_VEL
LIN {X 0,Y 131.191,Z 602.472,A -85,B 0,C 180,E1 -25973.894,E2 -25973.894} C_VEL
LIN {X 0,Y 124.721,Z 600.465,A -85,B 0,C 180,E1 -25979.526,E2 -25979.526} C_VEL
LIN {X 0,Y 119.898,Z 597.503,A -85,B 0,C 180,E1 -25985.775,E2 -25985.775} C_VEL
LIN {X 0,Y 117.142,Z 593.6,A -85,B 0,C 180,E1 -25992.544,E2 -25992.544} C_VEL
LIN {X 0,Y 116.393,Z 588.588,A -85,B 0,C 180,E1 -25999.563,E2 -25999.563} C_VEL
LIN {X 0,Y 117.444,Z 582.108,A -85,B 0,C 180,E1 -26006.569,E2 -26006.569} C_VEL
LIN {X 0,Y 118.347,Z 579.002,A -85,B 0,C 180,E1 -26009.362,E2 -26009.362} C_VEL
LIN {X 0,Y 116.897,Z 585.53,A -85,B 0,C 180,E1 -26015.174,E2 -26015.174} C_VEL
LIN {X 0,Y 116.351,Z 591.449,A -85,B 0,C 180,E1 -26022.205,E2 -26022.205} C_VEL
LIN {X 0,Y 117.583,Z 596.051,A -85,B 0,C 180,E1 -26029.192,E2 -26029.192} C_VEL
LIN {X 0,Y 119.881,Z 598.821,A -85,B 0,C 180,E1 -26034.228,E2 -26034.228} C_VEL
LIN {X 0,Y 124.661,Z 601.658,A -85,B 0,C 180,E1 -26040.49,E2 -26040.49} C_VEL
LIN {X 0,Y 131.119,Z 603.602,A -85,B 0,C 180,E1 -26046.129,E2 -26046.129} C_VEL
LIN {X 0,Y 139.122,Z 604.691,A -85,B 0,C 180,E1 -26051.05,E2 -26051.05} C_VEL
LIN {X 0,Y 150.832,Z 604.928,A -85,B 0,C 180,E1 -26056.082,E2 -26056.082} C_VEL
LIN {X 0,Y 152.077,Z 604.863,A -85,B 0,C 180,E1 -26056.528,E2 -26056.528} C_VEL
LIN {X 0,Y 152.348,Z 604.672,A -85,B 0,C 180,E1 -26057.427,E2 -26057.427} C_VEL
LIN {X 0,Y 144.208,Z 603.382,A -85,B 0,C 180,E1 -26060.687,E2 -26060.687} C_VEL
LIN {X 0,Y 135.405,Z 600.919,A -85,B 0,C 180,E1 -26065.185,E2 -26065.185} C_VEL
LIN {X 0,Y 126.38,Z 596.444,A -85,B 0,C 180,E1 -26071.792,E2 -26071.792} C_VEL
LIN {X 0,Y 120.89,Z 591.667,A -85,B 0,C 180,E1 -26077.798,E2 -26077.798} C_VEL
LIN {X 0,Y 116.791,Z 585.043,A -85,B 0,C 180,E1 -26084.913,E2 -26084.913} C_VEL
LIN {X 0,Y 115.118,Z 578.324,A -85,B 0,C 180,E1 -26091.222,E2 -26091.222} C_VEL
LIN {X 0,Y 114.423,Z 570.4,A -85,B 0,C 180,E1 -26097.355,E2 -26097.355} C_VEL
LIN {X 0,Y 114.123,Z 568.044,A -85,B 0,C 180,E1 -26098.917,E2 -26098.917} C_VEL
LIN {X 0,Y 112.864,Z 564.164,A -85,B 0,C 180,E1 -26101.084,E2 -26101.084} C_VEL
LIN {X 0,Y 108.602,Z 552.697,A -85,B 0,C 180,E1 -26106.456,E2 -26106.456} C_VEL
LIN {X 0,Y 108.257,Z 548.173,A -85,B 0,C 180,E1 -26108.537,E2 -26108.537} C_VEL
LIN {X 0,Y 109.333,Z 536.225,A -85,B 0,C 180,E1 -26113.588,E2 -26113.588} C_VEL
LIN {X 0,Y 110.653,Z 524.288,A -85,B 0,C 180,E1 -26117.69,E2 -26117.69} C_VEL
LIN {X 0,Y 110.58,Z 521.303,A -85,B 0,C 180,E1 -26118.53,E2 -26118.53} C_VEL
LIN {X 0,Y 107.936,Z 507.741,A -85,B 0,C 180,E1 -26121.737,E2 -26121.737} C_VEL
LIN {X 0,Y 107.107,Z 503.141,A -85,B 0,C 180,E1 -26122.809,E2 -26122.809} C_VEL
LIN {X 0,Y 107.12,Z 503.137,A -85,B 0,C 180,E1 -26131.661,E2 -26131.661} C_VEL
LIN {X 0,Y 107.436,Z 503.101,A -85,B 0,C 180,E1 -26136.069,E2 -26136.069} C_VEL
LIN {X 0,Y 107.564,Z 503.079,A -85,B 0,C 180,E1 -26140.798,E2 -26140.798} C_VEL
LIN {X 0,Y 107.668,Z 503.073,A -85,B 0,C 180,E1 -26145.893,E2 -26145.893} C_VEL
LIN {X 0,Y 107.709,Z 503.062,A -85,B 0,C 180,E1 -26151.538,E2 -26151.538} C_VEL
LIN {X 0,Y 107.81,Z 503.048,A -85,B 0,C 180,E1 -26158.566,E2 -26158.566} C_VEL
LIN {X 0,Y 107.914,Z 503.037,A -85,B 0,C 180,E1 -26166.998,E2 -26166.998} C_VEL
LIN {X 0,Y 108.043,Z 503.023,A -85,B 0,C 180,E1 -26174.918,E2 -26174.918} C_VEL
LIN {X 0,Y 108.31,Z 502.991,A -85,B 0,C 180,E1 -26178.775,E2 -26178.775} C_VEL
LIN {X 0,Y 108.466,Z 502.967,A -85,B 0,C 180,E1 -26186.285,E2 -26186.285} C_VEL
LIN {X 0,Y 108.946,Z 502.915,A -85,B 0,C 180,E1 -26190,E2 -26190} C_VEL
LIN {X 0,Y 108.306,Z 502.993,A -85,B 0,C 180,E1 -26197.457,E2 -26197.457} C_VEL
LIN {X 0,Y 108.176,Z 503.002,A -85,B 0,C 180,E1 -26202.955,E2 -26202.955} C_VEL
LIN {X 0,Y 107.907,Z 503.042,A -85,B 0,C 180,E1 -26209.005,E2 -26209.005} C_VEL
LIN {X 0,Y 107.861,Z 503.047,A -85,B 0,C 180,E1 -26214.184,E2 -26214.184} C_VEL
LIN {X 0,Y 107.798,Z 503.052,A -85,B 0,C 180,E1 -26222.051,E2 -26222.051} C_VEL
LIN {X 0,Y 107.71,Z 503.062,A -85,B 0,C 180,E1 -26228.463,E2 -26228.463} C_VEL
LIN {X 0,Y 107.667,Z 503.071,A -85,B 0,C 180,E1 -26235.892,E2 -26235.892} C_VEL
LIN {X 0,Y 107.601,Z 503.081,A -85,B 0,C 180,E1 -26241.609,E2 -26241.609} C_VEL
LIN {X 0,Y 107.499,Z 503.093,A -85,B 0,C 180,E1 -26243.955,E2 -26243.955} C_VEL
LIN {X 0,Y 107.207,Z 503.127,A -85,B 0,C 180,E1 -26248.454,E2 -26248.454} C_VEL
LIN {X 0,Y 107.158,Z 503.135,A -85,B 0,C 180,E1 -26258.097,E2 -26258.097} C_VEL
LIN {X 0,Y 109.728,Z 516.708,A -85,B 0,C 180,E1 -26261.079,E2 -26261.079} C_VEL
LIN {X 0,Y 110.729,Z 522.361,A -85,B 0,C 180,E1 -26262.531,E2 -26262.531} C_VEL
LIN {X 0,Y 109.377,Z 534.644,A -85,B 0,C 180,E1 -26266.609,E2 -26266.609} C_VEL
LIN {X 0,Y 108.413,Z 545.543,A -85,B 0,C 180,E1 -26271.142,E2 -26271.142} C_VEL
LIN {X 0,Y 107.85,Z 555.67,A -85,B 0,C 180,E1 -26276.263,E2 -26276.263} C_VEL
LIN {X 0,Y 107.765,Z 564.877,A -85,B 0,C 180,E1 -26281.868,E2 -26281.868} C_VEL
LIN {X 0,Y 108.331,Z 573.542,A -85,B 0,C 180,E1 -26288.393,E2 -26288.393} C_VEL
LIN {X 0,Y 109.763,Z 580.644,A -85,B 0,C 180,E1 -26294.839,E2 -26294.839} C_VEL
LIN {X 0,Y 113.211,Z 587.418,A -85,B 0,C 180,E1 -26301.867,E2 -26301.867} C_VEL
LIN {X 0,Y 118.444,Z 592.908,A -85,B 0,C 180,E1 -26308.338,E2 -26308.338} C_VEL
LIN {X 0,Y 125.503,Z 597.348,A -85,B 0,C 180,E1 -26314.054,E2 -26314.054} C_VEL
LIN {X 0,Y 133.879,Z 600.746,A -85,B 0,C 180,E1 -26319.045,E2 -26319.045} C_VEL
LIN {X 0,Y 141.997,Z 602.862,A -85,B 0,C 180,E1 -26322.659,E2 -26322.659} C_VEL
LIN {X 0,Y 140.869,Z 602.997,A -85,B 0,C 180,E1 -26323.973,E2 -26323.973} C_VEL
LIN {X 0,Y 129.657,Z 601.733,A -85,B 0,C 180,E1 -26329.424,E2 -26329.424} C_VEL
LIN {X 0,Y 122.049,Z 599.818,A -85,B 0,C 180,E1 -26334.842,E2 -26334.842} C_VEL
LIN {X 0,Y 116.138,Z 597.026,A -85,B 0,C 180,E1 -26341.045,E2 -26341.045} C_VEL
LIN {X 0,Y 112.019,Z 593.268,A -85,B 0,C 180,E1 -26347.887,E2 -26347.887} C_VEL
LIN {X 0,Y 110.177,Z 588.551,A -85,B 0,C 180,E1 -26355.217,E2 -26355.217} C_VEL
LIN {X 0,Y 110.35,Z 582.575,A -85,B 0,C 180,E1 -26362.682,E2 -26362.682} C_VEL
LIN {X 0,Y 112.056,Z 575.728,A -85,B 0,C 180,E1 -26369.326,E2 -26369.326} C_VEL
LIN {X 0,Y 110.511,Z 582.472,A -85,B 0,C 180,E1 -26375.474,E2 -26375.474} C_VEL
LIN {X 0,Y 109.945,Z 588.768,A -85,B 0,C 180,E1 -26382.928,E2 -26382.928} C_VEL
LIN {X 0,Y 112.003,Z 594.679,A -85,B 0,C 180,E1 -26392.116,E2 -26392.116} C_VEL
LIN {X 0,Y 116.073,Z 598.281,A -85,B 0,C 180,E1 -26398.972,E2 -26398.972} C_VEL
LIN {X 0,Y 122,Z 600.978,A -85,B 0,C 180,E1 -26405.175,E2 -26405.175} C_VEL
LIN {X 0,Y 129.549,Z 602.841,A -85,B 0,C 180,E1 -26410.617,E2 -26410.617} C_VEL
LIN {X 0,Y 140.827,Z 604.022,A -85,B 0,C 180,E1 -26416.115,E2 -26416.115} C_VEL
LIN {X 0,Y 141.942,Z 604.065,A -85,B 0,C 180,E1 -26416.553,E2 -26416.553} C_VEL
LIN {X 0,Y 140.984,Z 603.661,A -85,B 0,C 180,E1 -26417.899,E2 -26417.899} C_VEL
LIN {X 0,Y 129.668,Z 600.282,A -85,B 0,C 180,E1 -26423.403,E2 -26423.403} C_VEL
LIN {X 0,Y 120.269,Z 595.3,A -85,B 0,C 180,E1 -26430.219,E2 -26430.219} C_VEL
LIN {X 0,Y 114.514,Z 590.106,A -85,B 0,C 180,E1 -26436.49,E2 -26436.49} C_VEL
LIN {X 0,Y 110.696,Z 584.295,A -85,B 0,C 180,E1 -26442.786,E2 -26442.786} C_VEL
LIN {X 0,Y 108.616,Z 577.081,A -85,B 0,C 180,E1 -26449.751,E2 -26449.751} C_VEL
LIN {X 0,Y 107.815,Z 570.236,A -85,B 0,C 180,E1 -26455.327,E2 -26455.327} C_VEL
LIN {X 0,Y 107.662,Z 562.065,A -85,B 0,C 180,E1 -26460.936,E2 -26460.936} C_VEL
LIN {X 0,Y 107.902,Z 554.013,A -85,B 0,C 180,E1 -26465.608,E2 -26465.608} C_VEL
LIN {X 0,Y 108.257,Z 548.173,A -85,B 0,C 180,E1 -26468.537,E2 -26468.537} C_VEL
LIN {X 0,Y 108.216,Z 543.651,A -85,B 0,C 180,E1 -26470.515,E2 -26470.515} C_VEL
LIN {X 0,Y 107.533,Z 538.851,A -85,B 0,C 180,E1 -26472.347,E2 -26472.347} C_VEL
LIN {X 0,Y 105.193,Z 528.826,A -85,B 0,C 180,E1 -26475.631,E2 -26475.631} C_VEL
LIN {X 0,Y 103.646,Z 521.802,A -85,B 0,C 180,E1 -26477.664,E2 -26477.664} C_VEL
LIN {X 0,Y 100.904,Z 507.915,A -85,B 0,C 180,E1 -26481.153,E2 -26481.153} C_VEL
LIN {X 0,Y 100.172,Z 504.006,A -85,B 0,C 180,E1 -26482.129,E2 -26482.129} C_VEL
LIN {X 0,Y 100.098,Z 504.008,A -85,B 0,C 180,E1 -26492.591,E2 -26492.591} C_VEL
LIN {X 0,Y 100.486,Z 503.965,A -85,B 0,C 180,E1 -26499.705,E2 -26499.705} C_VEL
LIN {X 0,Y 100.634,Z 503.949,A -85,B 0,C 180,E1 -26505.703,E2 -26505.703} C_VEL
LIN {X 0,Y 100.647,Z 503.941,A -85,B 0,C 180,E1 -26511.063,E2 -26511.063} C_VEL
LIN {X 0,Y 100.703,Z 503.938,A -85,B 0,C 180,E1 -26516.877,E2 -26516.877} C_VEL
LIN {X 0,Y 100.789,Z 503.929,A -85,B 0,C 180,E1 -26525.268,E2 -26525.268} C_VEL
LIN {X 0,Y 100.822,Z 503.921,A -85,B 0,C 180,E1 -26529.602,E2 -26529.602} C_VEL
LIN {X 0,Y 101.203,Z 503.872,A -85,B 0,C 180,E1 -26537.975,E2 -26537.975} C_VEL
LIN {X 0,Y 101.283,Z 503.869,A -85,B 0,C 180,E1 -26542.023,E2 -26542.023} C_VEL
LIN {X 0,Y 101.869,Z 503.797,A -85,B 0,C 180,E1 -26550,E2 -26550} C_VEL
LIN {X 0,Y 101.244,Z 503.874,A -85,B 0,C 180,E1 -26557.98,E2 -26557.98} C_VEL
LIN {X 0,Y 101.105,Z 503.882,A -85,B 0,C 180,E1 -26563.297,E2 -26563.297} C_VEL
LIN {X 0,Y 100.819,Z 503.922,A -85,B 0,C 180,E1 -26570.398,E2 -26570.398} C_VEL
LIN {X 0,Y 100.777,Z 503.93,A -85,B 0,C 180,E1 -26574.958,E2 -26574.958} C_VEL
LIN {X 0,Y 100.703,Z 503.938,A -85,B 0,C 180,E1 -26583.123,E2 -26583.123} C_VEL
LIN {X 0,Y 100.656,Z 503.939,A -85,B 0,C 180,E1 -26589.82,E2 -26589.82} C_VEL
LIN {X 0,Y 100.64,Z 503.947,A -85,B 0,C 180,E1 -26595.705,E2 -26595.705} C_VEL
LIN {X 0,Y 100.553,Z 503.958,A -85,B 0,C 180,E1 -26601.019,E2 -26601.019} C_VEL
LIN {X 0,Y 100.189,Z 503.997,A -85,B 0,C 180,E1 -26607.328,E2 -26607.328} C_VEL
LIN {X 0,Y 100.22,Z 503.997,A -85,B 0,C 180,E1 -26618.756,E2 -26618.756} C_VEL
LIN {X 0,Y 103.22,Z 519.132,A -85,B 0,C 180,E1 -26622.408,E2 -26622.408} C_VEL
LIN {X 0,Y 103.711,Z 521.973,A -85,B 0,C 180,E1 -26623.193,E2 -26623.193} C_VEL
LIN {X 0,Y 102.419,Z 534.269,A -85,B 0,C 180,E1 -26627.616,E2 -26627.616} C_VEL
LIN {X 0,Y 101.604,Z 544.375,A -85,B 0,C 180,E1 -26632.047,E2 -26632.047} C_VEL
LIN {X 0,Y 101.132,Z 553.818,A -85,B 0,C 180,E1 -26637.011,E2 -26637.011} C_VEL
LIN {X 0,Y 101.184,Z 563.128,A -85,B 0,C 180,E1 -26642.985,E2 -26642.985} C_VEL
LIN {X 0,Y 101.901,Z 572.065,A -85,B 0,C 180,E1 -26649.928,E2 -26649.928} C_VEL
LIN {X 0,Y 104.25,Z 580.896,A -85,B 0,C 180,E1 -26658.307,E2 -26658.307} C_VEL
LIN {X 0,Y 109.456,Z 588.607,A -85,B 0,C 180,E1 -26666.708,E2 -26666.708} C_VEL
LIN {X 0,Y 115.872,Z 593.943,A -85,B 0,C 180,E1 -26673.084,E2 -26673.084} C_VEL
LIN {X 0,Y 123.912,Z 598.248,A -85,B 0,C 180,E1 -26678.6,E2 -26678.6} C_VEL
LIN {X 0,Y 131.947,Z 601.166,A -85,B 0,C 180,E1 -26682.642,E2 -26682.642} C_VEL
LIN {X 0,Y 130.992,Z 601.229,A -85,B 0,C 180,E1 -26684.025,E2 -26684.025} C_VEL
LIN {X 0,Y 124.484,Z 600.107,A -85,B 0,C 180,E1 -26687.352,E2 -26687.352} C_VEL
LIN {X 0,Y 116.536,Z 597.832,A -85,B 0,C 180,E1 -26692.909,E2 -26692.909} C_VEL
LIN {X 0,Y 110.297,Z 594.738,A -85,B 0,C 180,E1 -26699.353,E2 -26699.353} C_VEL
LIN {X 0,Y 105.928,Z 590.704,A -85,B 0,C 180,E1 -26706.541,E2 -26706.541} C_VEL
LIN {X 0,Y 103.901,Z 585.713,A -85,B 0,C 180,E1 -26714.302,E2 -26714.302} C_VEL
LIN {X 0,Y 104.059,Z 579.388,A -85,B 0,C 180,E1 -26722.237,E2 -26722.237} C_VEL
LIN {X 0,Y 105.839,Z 572.326,A -85,B 0,C 180,E1 -26729.358,E2 -26729.358} C_VEL
LIN {X 0,Y 104.202,Z 579.248,A -85,B 0,C 180,E1 -26735.806,E2 -26735.806} C_VEL
LIN {X 0,Y 103.61,Z 584.329,A -85,B 0,C 180,E1 -26741.741,E2 -26741.741} C_VEL
LIN {X 0,Y 104.606,Z 589.949,A -85,B 0,C 180,E1 -26749.85,E2 -26749.85} C_VEL
LIN {X 0,Y 107.784,Z 594.179,A -85,B 0,C 180,E1 -26757.157,E2 -26757.157} C_VEL
LIN {X 0,Y 113.137,Z 597.639,A -85,B 0,C 180,E1 -26763.992,E2 -26763.992} C_VEL
LIN {X 0,Y 120.245,Z 600.232,A -85,B 0,C 180,E1 -26770.01,E2 -26770.01} C_VEL
LIN {X 0,Y 130.977,Z 602.299,A -85,B 0,C 180,E1 -26776.066,E2 -26776.066} C_VEL
LIN {X 0,Y 132.065,Z 602.246,A -85,B 0,C 180,E1 -26777.473,E2 -26777.473} C_VEL
LIN {X 0,Y 124.093,Z 599.401,A -85,B 0,C 180,E1 -26781.466,E2 -26781.466} C_VEL
LIN {X 0,Y 116.006,Z 595.144,A -85,B 0,C 180,E1 -26786.959,E2 -26786.959} C_VEL
LIN {X 0,Y 109.588,Z 589.902,A -85,B 0,C 180,E1 -26793.327,E2 -26793.327} C_VEL
LIN {X 0,Y 104.244,Z 582.206,A -85,B 0,C 180,E1 -26801.665,E2 -26801.665} C_VEL
LIN {X 0,Y 102.041,Z 574.578,A -85,B 0,C 180,E1 -26809.083,E2 -26809.083} C_VEL
LIN {X 0,Y 101.115,Z 566.125,A -85,B 0,C 180,E1 -26816.015,E2 -26816.015} C_VEL
LIN {X 0,Y 101.017,Z 557.169,A -85,B 0,C 180,E1 -26821.994,E2 -26821.994} C_VEL
LIN {X 0,Y 101.512,Z 546.305,A -85,B 0,C 180,E1 -26827.96,E2 -26827.96} C_VEL
LIN {X 0,Y 102.388,Z 535.344,A -85,B 0,C 180,E1 -26832.891,E2 -26832.891} C_VEL
LIN {X 0,Y 103.664,Z 523.382,A -85,B 0,C 180,E1 -26837.19,E2 -26837.19} C_VEL
LIN {X 0,Y 103.646,Z 521.802,A -85,B 0,C 180,E1 -26837.664,E2 -26837.664} C_VEL
LIN {X 0,Y 102.584,Z 519.943,A -85,B 0,C 180,E1 -26838.111,E2 -26838.111} C_VEL
LIN {X 0,Y 95.786,Z 514.966,A -85,B 0,C 180,E1 -26838.785,E2 -26838.785} C_VEL
LIN {X 0,Y 94.915,Z 513.338,A -85,B 0,C 180,E1 -26839.127,E2 -26839.127} C_VEL
LIN {X 0,Y 93.296,Z 504.865,A -85,B 0,C 180,E1 -26841.199,E2 -26841.199} C_VEL
LIN {X 0,Y 93.111,Z 504.879,A -85,B 0,C 180,E1 -26853.872,E2 -26853.872} C_VEL
LIN {X 0,Y 93.417,Z 504.84,A -85,B 0,C 180,E1 -26861.208,E2 -26861.208} C_VEL
LIN {X 0,Y 93.541,Z 504.829,A -85,B 0,C 180,E1 -26868.707,E2 -26868.707} C_VEL
LIN {X 0,Y 93.601,Z 504.826,A -85,B 0,C 180,E1 -26875.685,E2 -26875.685} C_VEL
LIN {X 0,Y 93.672,Z 504.817,A -85,B 0,C 180,E1 -26884.205,E2 -26884.205} C_VEL
LIN {X 0,Y 93.697,Z 504.806,A -85,B 0,C 180,E1 -26887.973,E2 -26887.973} C_VEL
LIN {X 0,Y 94.101,Z 504.755,A -85,B 0,C 180,E1 -26897.053,E2 -26897.053} C_VEL
LIN {X 0,Y 94.215,Z 504.749,A -85,B 0,C 180,E1 -26901.42,E2 -26901.42} C_VEL
LIN {X 0,Y 94.794,Z 504.678,A -85,B 0,C 180,E1 -26910,E2 -26910} C_VEL
LIN {X 0,Y 94.178,Z 504.754,A -85,B 0,C 180,E1 -26918.583,E2 -26918.583} C_VEL
LIN {X 0,Y 94.025,Z 504.764,A -85,B 0,C 180,E1 -26923.658,E2 -26923.658} C_VEL
LIN {X 0,Y 93.695,Z 504.806,A -85,B 0,C 180,E1 -26932.027,E2 -26932.027} C_VEL
LIN {X 0,Y 93.626,Z 504.822,A -85,B 0,C 180,E1 -26936.769,E2 -26936.769} C_VEL
LIN {X 0,Y 93.601,Z 504.826,A -85,B 0,C 180,E1 -26944.315,E2 -26944.315} C_VEL
LIN {X 0,Y 93.537,Z 504.833,A -85,B 0,C 180,E1 -26952.55,E2 -26952.55} C_VEL
LIN {X 0,Y 93.499,Z 504.83,A -85,B 0,C 180,E1 -26958.735,E2 -26958.735} C_VEL
LIN {X 0,Y 93.197,Z 504.869,A -85,B 0,C 180,E1 -26966.049,E2 -26966.049} C_VEL
LIN {X 0,Y 92.834,Z 504.914,A -85,B 0,C 180,E1 -26975.293,E2 -26975.293} C_VEL
LIN {X 0,Y 93.413,Z 504.988,A -85,B 0,C 180,E1 -26979.782,E2 -26979.782} C_VEL
LIN {X 0,Y 96.248,Z 518.866,A -85,B 0,C 180,E1 -26983.29,E2 -26983.29} C_VEL
LIN {X 0,Y 96.67,Z 521.873,A -85,B 0,C 180,E1 -26984.178,E2 -26984.178} C_VEL
LIN {X 0,Y 95.494,Z 534.032,A -85,B 0,C 180,E1 -26988.86,E2 -26988.86} C_VEL
LIN {X 0,Y 94.792,Z 544.06,A -85,B 0,C 180,E1 -26993.614,E2 -26993.614} C_VEL
LIN {X 0,Y 94.487,Z 553.37,A -85,B 0,C 180,E1 -26998.933,E2 -26998.933} C_VEL
LIN {X 0,Y 94.671,Z 561.305,A -85,B 0,C 180,E1 -27004.256,E2 -27004.256} C_VEL
LIN {X 0,Y 95.438,Z 569.199,A -85,B 0,C 180,E1 -27010.608,E2 -27010.608} C_VEL
LIN {X 0,Y 97.606,Z 577.88,A -85,B 0,C 180,E1 -27018.905,E2 -27018.905} C_VEL
LIN {X 0,Y 101.96,Z 585.081,A -85,B 0,C 180,E1 -27026.615,E2 -27026.615} C_VEL
LIN {X 0,Y 110.134,Z 592.414,A -85,B 0,C 180,E1 -27035.051,E2 -27035.051} C_VEL
LIN {X 0,Y 118.529,Z 597.094,A -85,B 0,C 180,E1 -27040.709,E2 -27040.709} C_VEL
LIN {X 0,Y 123.052,Z 599.047,A -85,B 0,C 180,E1 -27043.264,E2 -27043.264} C_VEL
LIN {X 0,Y 115.193,Z 597.07,A -85,B 0,C 180,E1 -27047.847,E2 -27047.847} C_VEL
LIN {X 0,Y 107.703,Z 594.074,A -85,B 0,C 180,E1 -27054.036,E2 -27054.036} C_VEL
LIN {X 0,Y 102.007,Z 590.205,A -85,B 0,C 180,E1 -27061.165,E2 -27061.165} C_VEL
LIN {X 0,Y 98.579,Z 585.43,A -85,B 0,C 180,E1 -27069.117,E2 -27069.117} C_VEL
LIN {X 0,Y 97.558,Z 579.552,A -85,B 0,C 180,E1 -27077.519,E2 -27077.519} C_VEL
LIN {X 0,Y 98.681,Z 572.085,A -85,B 0,C 180,E1 -27085.916,E2 -27085.916} C_VEL
LIN {X 0,Y 99.766,Z 568.645,A -85,B 0,C 180,E1 -27089.369,E2 -27089.369} C_VEL
LIN {X 0,Y 97.969,Z 575.868,A -85,B 0,C 180,E1 -27096.177,E2 -27096.177} C_VEL
LIN {X 0,Y 97.408,Z 581.148,A -85,B 0,C 180,E1 -27102.501,E2 -27102.501} C_VEL
LIN {X 0,Y 98.477,Z 586.942,A -85,B 0,C 180,E1 -27110.906,E2 -27110.906} C_VEL
LIN {X 0,Y 101.943,Z 591.618,A -85,B 0,C 180,E1 -27118.854,E2 -27118.854} C_VEL
LIN {X 0,Y 107.643,Z 595.342,A -85,B 0,C 180,E1 -27125.988,E2 -27125.988} C_VEL
LIN {X 0,Y 115.107,Z 598.218,A -85,B 0,C 180,E1 -27132.192,E2 -27132.192} C_VEL
LIN {X 0,Y 121.776,Z 599.901,A -85,B 0,C 180,E1 -27136.169,E2 -27136.169} C_VEL
LIN {X 0,Y 122.227,Z 599.783,A -85,B 0,C 180,E1 -27137.498,E2 -27137.498} C_VEL
LIN {X 0,Y 112.256,Z 594.898,A -85,B 0,C 180,E1 -27143.505,E2 -27143.505} C_VEL
LIN {X 0,Y 103.513,Z 588,A -85,B 0,C 180,E1 -27151.624,E2 -27151.624} C_VEL
LIN {X 0,Y 98.52,Z 581.151,A -85,B 0,C 180,E1 -27159.104,E2 -27159.104} C_VEL
LIN {X 0,Y 95.77,Z 573.052,A -85,B 0,C 180,E1 -27167.283,E2 -27167.283} C_VEL
LIN {X 0,Y 94.634,Z 564.266,A -85,B 0,C 180,E1 -27174.674,E2 -27174.674} C_VEL
LIN {X 0,Y 94.402,Z 555.229,A -85,B 0,C 180,E1 -27181.067,E2 -27181.067} C_VEL
LIN {X 0,Y 94.818,Z 543.995,A -85,B 0,C 180,E1 -27187.454,E2 -27187.454} C_VEL
LIN {X 0,Y 95.831,Z 531.311,A -85,B 0,C 180,E1 -27193.25,E2 -27193.25} C_VEL
LIN {X 0,Y 96.647,Z 523.063,A -85,B 0,C 180,E1 -27196.368,E2 -27196.368} C_VEL
LIN {X 0,Y 96.285,Z 519.895,A -85,B 0,C 180,E1 -27197.357,E2 -27197.357} C_VEL
LIN {X 0,Y 94.915,Z 513.338,A -85,B 0,C 180,E1 -27199.127,E2 -27199.127} C_VEL
LIN {X 0,Y 93.87,Z 510.373,A -85,B 0,C 180,E1 -27200.343,E2 -27200.343} C_VEL
LIN {X 0,Y 92.452,Z 508.25,A -85,B 0,C 180,E1 -27202.056,E2 -27202.056} C_VEL
LIN {X 0,Y 90.16,Z 506.363,A -85,B 0,C 180,E1 -27205.229,E2 -27205.229} C_VEL
LIN {X 0,Y 88.06,Z 505.702,A -85,B 0,C 180,E1 -27209.008,E2 -27209.008} C_VEL
LIN {X 0,Y 86.293,Z 505.731,A -85,B 0,C 180,E1 -27214.568,E2 -27214.568} C_VEL
LIN {X 0,Y 86.103,Z 505.744,A -85,B 0,C 180,E1 -27217.437,E2 -27217.437} C_VEL
LIN {X 0,Y 86.382,Z 505.719,A -85,B 0,C 180,E1 -27222.926,E2 -27222.926} C_VEL
LIN {X 0,Y 86.464,Z 505.708,A -85,B 0,C 180,E1 -27229.438,E2 -27229.438} C_VEL
LIN {X 0,Y 86.545,Z 505.704,A -85,B 0,C 180,E1 -27235.358,E2 -27235.358} C_VEL
LIN {X 0,Y 86.588,Z 505.699,A -85,B 0,C 180,E1 -27243.234,E2 -27243.234} C_VEL
LIN {X 0,Y 86.667,Z 505.688,A -85,B 0,C 180,E1 -27251.073,E2 -27251.073} C_VEL
LIN {X 0,Y 86.972,Z 505.644,A -85,B 0,C 180,E1 -27255.97,E2 -27255.97} C_VEL
LIN {X 0,Y 87.121,Z 505.633,A -85,B 0,C 180,E1 -27260.715,E2 -27260.715} C_VEL
LIN {X 0,Y 87.721,Z 505.559,A -85,B 0,C 180,E1 -27270,E2 -27270} C_VEL
LIN {X 0,Y 87.087,Z 505.637,A -85,B 0,C 180,E1 -27279.288,E2 -27279.288} C_VEL
LIN {X 0,Y 86.934,Z 505.648,A -85,B 0,C 180,E1 -27284.036,E2 -27284.036} C_VEL
LIN {X 0,Y 86.648,Z 505.691,A -85,B 0,C 180,E1 -27288.932,E2 -27288.932} C_VEL
LIN {X 0,Y 86.588,Z 505.699,A -85,B 0,C 180,E1 -27296.766,E2 -27296.766} C_VEL
LIN {X 0,Y 86.52,Z 505.708,A -85,B 0,C 180,E1 -27305.676,E2 -27305.676} C_VEL
LIN {X 0,Y 86.458,Z 505.715,A -85,B 0,C 180,E1 -27312.978,E2 -27312.978} C_VEL
LIN {X 0,Y 86.399,Z 505.716,A -85,B 0,C 180,E1 -27319.4,E2 -27319.4} C_VEL
LIN {X 0,Y 86.158,Z 505.748,A -85,B 0,C 180,E1 -27325.179,E2 -27325.179} C_VEL
LIN {X 0,Y 85.811,Z 505.787,A -85,B 0,C 180,E1 -27335.825,E2 -27335.825} C_VEL
LIN {X 0,Y 86.552,Z 505.702,A -85,B 0,C 180,E1 -27340.815,E2 -27340.815} C_VEL
LIN {X 0,Y 89.559,Z 519.74,A -85,B 0,C 180,E1 -27344.653,E2 -27344.653} C_VEL
LIN {X 0,Y 89.47,Z 524.451,A -85,B 0,C 180,E1 -27346.369,E2 -27346.369} C_VEL
LIN {X 0,Y 88.465,Z 537.123,A -85,B 0,C 180,E1 -27352.007,E2 -27352.007} C_VEL
LIN {X 0,Y 88.008,Z 547.495,A -85,B 0,C 180,E1 -27357.711,E2 -27357.711} C_VEL
LIN {X 0,Y 88.13,Z 556.177,A -85,B 0,C 180,E1 -27363.428,E2 -27363.428} C_VEL
LIN {X 0,Y 88.842,Z 564.804,A -85,B 0,C 180,E1 -27370.252,E2 -27370.252} C_VEL
LIN {X 0,Y 90.26,Z 571.997,A -85,B 0,C 180,E1 -27376.976,E2 -27376.976} C_VEL
LIN {X 0,Y 94.644,Z 581.042,A -85,B 0,C 180,E1 -27386.457,E2 -27386.457} C_VEL
LIN {X 0,Y 102.622,Z 589.188,A -85,B 0,C 180,E1 -27395.599,E2 -27395.599} C_VEL
LIN {X 0,Y 113.348,Z 595.72,A -85,B 0,C 180,E1 -27403.003,E2 -27403.003} C_VEL
LIN {X 0,Y 110.295,Z 594.847,A -85,B 0,C 180,E1 -27405.499,E2 -27405.499} C_VEL
LIN {X 0,Y 102.403,Z 591.555,A -85,B 0,C 180,E1 -27411.853,E2 -27411.853} C_VEL
LIN {X 0,Y 96.341,Z 587.412,A -85,B 0,C 180,E1 -27419.293,E2 -27419.293} C_VEL
LIN {X 0,Y 92.103,Z 580.909,A -85,B 0,C 180,E1 -27429.917,E2 -27429.917} C_VEL
LIN {X 0,Y 91.557,Z 574.377,A -85,B 0,C 180,E1 -27438.936,E2 -27438.936} C_VEL
LIN {X 0,Y 92.956,Z 567.052,A -85,B 0,C 180,E1 -27446.916,E2 -27446.916} C_VEL
LIN {X 0,Y 93.829,Z 564.775,A -85,B 0,C 180,E1 -27449.329,E2 -27449.329} C_VEL
LIN {X 0,Y 91.92,Z 571.973,A -85,B 0,C 180,E1 -27456.311,E2 -27456.311} C_VEL
LIN {X 0,Y 91.319,Z 577.811,A -85,B 0,C 180,E1 -27463.349,E2 -27463.349} C_VEL
LIN {X 0,Y 92.545,Z 583.854,A -85,B 0,C 180,E1 -27472.316,E2 -27472.316} C_VEL
LIN {X 0,Y 96.276,Z 588.818,A -85,B 0,C 180,E1 -27480.73,E2 -27480.73} C_VEL
LIN {X 0,Y 102.331,Z 592.871,A -85,B 0,C 180,E1 -27488.179,E2 -27488.179} C_VEL
LIN {X 0,Y 110.206,Z 596.023,A -85,B 0,C 180,E1 -27494.547,E2 -27494.547} C_VEL
LIN {X 0,Y 113.489,Z 596.958,A -85,B 0,C 180,E1 -27497.064,E2 -27497.064} C_VEL
LIN {X 0,Y 102.793,Z 590.509,A -85,B 0,C 180,E1 -27504.469,E2 -27504.469} C_VEL
LIN {X 0,Y 94.679,Z 582.421,A -85,B 0,C 180,E1 -27513.553,E2 -27513.553} C_VEL
LIN {X 0,Y 90.584,Z 574.574,A -85,B 0,C 180,E1 -27521.921,E2 -27521.921} C_VEL
LIN {X 0,Y 88.682,Z 566.43,A -85,B 0,C 180,E1 -27529.73,E2 -27529.73} C_VEL
LIN {X 0,Y 88.008,Z 557.901,A -85,B 0,C 180,E1 -27536.567,E2 -27536.567} C_VEL
LIN {X 0,Y 87.904,Z 547.526,A -85,B 0,C 180,E1 -27543.439,E2 -27543.439} C_VEL
LIN {X 0,Y 88.337,Z 538.171,A -85,B 0,C 180,E1 -27548.58,E2 -27548.58} C_VEL
LIN {X 0,Y 89.416,Z 525.545,A -85,B 0,C 180,E1 -27554.22,E2 -27554.22} C_VEL
LIN {X 0,Y 89.631,Z 520.915,A -85,B 0,C 180,E1 -27555.93,E2 -27555.93} C_VEL
LIN {X 0,Y 86.591,Z 506.258,A -85,B 0,C 180,E1 -27559.975,E2 -27559.975} C_VEL
LIN {X 0,Y 86.417,Z 505.722,A -85,B 0,C 180,E1 -27560.222,E2 -27560.222} C_VEL
LIN {X 0,Y 85.749,Z 505.803,A -85,B 0,C 180,E1 -27569.458,E2 -27569.458} C_VEL
LIN {X 0,Y 86.099,Z 505.758,A -85,B 0,C 180,E1 -27575.287,E2 -27575.287} C_VEL
LIN {X 0,Y 86.103,Z 505.744,A -85,B 0,C 180,E1 -27577.437,E2 -27577.437} C_VEL
LIN {X 0,Y 85.861,Z 505.784,A -85,B 0,C 180,E1 -27580.05,E2 -27580.05} C_VEL
LIN {X 0,Y 84.617,Z 505.941,A -85,B 0,C 180,E1 -27583.942,E2 -27583.942} C_VEL
LIN {X 0,Y 81.566,Z 506.325,A -85,B 0,C 180,E1 -27590.554,E2 -27590.554} C_VEL
LIN {X 0,Y 79.668,Z 506.56,A -85,B 0,C 180,E1 -27596.211,E2 -27596.211} C_VEL
LIN {X 0,Y 79.371,Z 506.587,A -85,B 0,C 180,E1 -27599.145,E2 -27599.145} C_VEL
LIN {X 0,Y 79.528,Z 506.579,A -85,B 0,C 180,E1 -27603.778,E2 -27603.778} C_VEL
LIN {X 0,Y 79.526,Z 506.572,A -85,B 0,C 180,E1 -27609.299,E2 -27609.299} C_VEL
LIN {X 0,Y 79.845,Z 506.533,A -85,B 0,C 180,E1 -27615.525,E2 -27615.525} C_VEL
LIN {X 0,Y 80.004,Z 506.518,A -85,B 0,C 180,E1 -27619.881,E2 -27619.881} C_VEL
LIN {X 0,Y 80.647,Z 506.44,A -85,B 0,C 180,E1 -27630,E2 -27630} C_VEL
LIN {X 0,Y 79.97,Z 506.522,A -85,B 0,C 180,E1 -27640.123,E2 -27640.123} C_VEL
LIN {X 0,Y 79.747,Z 506.548,A -85,B 0,C 180,E1 -27645.331,E2 -27645.331} C_VEL
LIN {X 0,Y 79.516,Z 506.574,A -85,B 0,C 180,E1 -27650.704,E2 -27650.704} C_VEL
LIN {X 0,Y 79.486,Z 506.582,A -85,B 0,C 180,E1 -27657.846,E2 -27657.846} C_VEL
LIN {X 0,Y 79.387,Z 506.589,A -85,B 0,C 180,E1 -27662.085,E2 -27662.085} C_VEL
LIN {X 0,Y 79.374,Z 506.591,A -85,B 0,C 180,E1 -27668.302,E2 -27668.302} C_VEL
LIN {X 0,Y 79.35,Z 506.6,A -85,B 0,C 180,E1 -27675.118,E2 -27675.118} C_VEL
LIN {X 0,Y 79.123,Z 506.629,A -85,B 0,C 180,E1 -27683.075,E2 -27683.075} C_VEL
LIN {X 0,Y 78.843,Z 506.655,A -85,B 0,C 180,E1 -27687.665,E2 -27687.665} C_VEL
LIN {X 0,Y 79.838,Z 506.541,A -85,B 0,C 180,E1 -27702.273,E2 -27702.273} C_VEL
LIN {X 0,Y 82.597,Z 518.855,A -85,B 0,C 180,E1 -27705.839,E2 -27705.839} C_VEL
LIN {X 0,Y 82.874,Z 520.834,A -85,B 0,C 180,E1 -27706.513,E2 -27706.513} C_VEL
LIN {X 0,Y 81.933,Z 532.971,A -85,B 0,C 180,E1 -27711.986,E2 -27711.986} C_VEL
LIN {X 0,Y 81.563,Z 542.961,A -85,B 0,C 180,E1 -27717.53,E2 -27717.53} C_VEL
LIN {X 0,Y 81.798,Z 553.848,A -85,B 0,C 180,E1 -27724.928,E2 -27724.928} C_VEL
LIN {X 0,Y 82.738,Z 562.754,A -85,B 0,C 180,E1 -27732.259,E2 -27732.259} C_VEL
LIN {X 0,Y 84.854,Z 571.206,A -85,B 0,C 180,E1 -27740.609,E2 -27740.609} C_VEL
LIN {X 0,Y 89.704,Z 579.663,A -85,B 0,C 180,E1 -27749.739,E2 -27749.739} C_VEL
LIN {X 0,Y 97.193,Z 587.026,A -85,B 0,C 180,E1 -27757.924,E2 -27757.924} C_VEL
LIN {X 0,Y 103.685,Z 591.481,A -85,B 0,C 180,E1 -27762.673,E2 -27762.673} C_VEL
LIN {X 0,Y 103.997,Z 591.84,A -85,B 0,C 180,E1 -27764.051,E2 -27764.051} C_VEL
LIN {X 0,Y 93.872,Z 586.718,A -85,B 0,C 180,E1 -27773.206,E2 -27773.206} C_VEL
LIN {X 0,Y 88.529,Z 581.825,A -85,B 0,C 180,E1 -27781.555,E2 -27781.555} C_VEL
LIN {X 0,Y 85.851,Z 575.963,A -85,B 0,C 180,E1 -27790.886,E2 -27790.886} C_VEL
LIN {X 0,Y 85.852,Z 568.718,A -85,B 0,C 180,E1 -27800.577,E2 -27800.577} C_VEL
LIN {X 0,Y 88.047,Z 560.65,A -85,B 0,C 180,E1 -27809.186,E2 -27809.186} C_VEL
LIN {X 0,Y 86.26,Z 566.185,A -85,B 0,C 180,E1 -27814.673,E2 -27814.673} C_VEL
LIN {X 0,Y 85.442,Z 572.465,A -85,B 0,C 180,E1 -27821.864,E2 -27821.864} C_VEL
LIN {X 0,Y 86.157,Z 579.097,A -85,B 0,C 180,E1 -27831.535,E2 -27831.535} C_VEL
LIN {X 0,Y 89.181,Z 584.158,A -85,B 0,C 180,E1 -27839.905,E2 -27839.905} C_VEL
LIN {X 0,Y 95.46,Z 589.154,A -85,B 0,C 180,E1 -27848.741,E2 -27848.741} C_VEL
LIN {X 0,Y 104.011,Z 593.091,A -85,B 0,C 180,E1 -27856.042,E2 -27856.042} C_VEL
LIN {X 0,Y 103.81,Z 592.782,A -85,B 0,C 180,E1 -27857.391,E2 -27857.391} C_VEL
LIN {X 0,Y 93.803,Z 585.447,A -85,B 0,C 180,E1 -27865.503,E2 -27865.503} C_VEL
LIN {X 0,Y 87.435,Z 577.895,A -85,B 0,C 180,E1 -27873.764,E2 -27873.764} C_VEL
LIN {X 0,Y 83.744,Z 569.353,A -85,B 0,C 180,E1 -27882.92,E2 -27882.92} C_VEL
LIN {X 0,Y 81.997,Z 560.221,A -85,B 0,C 180,E1 -27891.375,E2 -27891.375} C_VEL
LIN {X 0,Y 81.484,Z 552.355,A -85,B 0,C 180,E1 -27897.53,E2 -27897.53} C_VEL
LIN {X 0,Y 81.426,Z 542.904,A -85,B 0,C 180,E1 -27903.713,E2 -27903.713} C_VEL
LIN {X 0,Y 81.965,Z 531.622,A -85,B 0,C 180,E1 -27909.876,E2 -27909.876} C_VEL
LIN {X 0,Y 82.757,Z 522.131,A -85,B 0,C 180,E1 -27914.133,E2 -27914.133} C_VEL
LIN {X 0,Y 82.219,Z 518.49,A -85,B 0,C 180,E1 -27915.371,E2 -27915.371} C_VEL
LIN {X 0,Y 79.635,Z 506.566,A -85,B 0,C 180,E1 -27918.954,E2 -27918.954} C_VEL
LIN {X 0,Y 78.787,Z 506.662,A -85,B 0,C 180,E1 -27932.36,E2 -27932.36} C_VEL
LIN {X 0,Y 79.111,Z 506.63,A -85,B 0,C 180,E1 -27938.454,E2 -27938.454} C_VEL
LIN {X 0,Y 79.33,Z 506.603,A -85,B 0,C 180,E1 -27945.134,E2 -27945.134} C_VEL
LIN {X 0,Y 79.395,Z 506.592,A -85,B 0,C 180,E1 -27952.816,E2 -27952.816} C_VEL
LIN {X 0,Y 79.371,Z 506.587,A -85,B 0,C 180,E1 -27959.145,E2 -27959.145} C_VEL
LIN {X 0,Y 79.068,Z 506.634,A -85,B 0,C 180,E1 -27961.979,E2 -27961.979} C_VEL
LIN {X 0,Y 77.78,Z 506.797,A -85,B 0,C 180,E1 -27966.204,E2 -27966.204} C_VEL
LIN {X 0,Y 74.786,Z 507.169,A -85,B 0,C 180,E1 -27973.418,E2 -27973.418} C_VEL
LIN {X 0,Y 73.077,Z 507.38,A -85,B 0,C 180,E1 -27979.61,E2 -27979.61} C_VEL
LIN {X 0,Y 72.93,Z 507.385,A -85,B 0,C 180,E1 -27982.807,E2 -27982.807} C_VEL
LIN {X 0,Y 73.573,Z 507.321,A -85,B 0,C 180,E1 -27990,E2 -27990} C_VEL
LIN {X 0,Y 72.861,Z 507.405,A -85,B 0,C 180,E1 -28001.123,E2 -28001.123} C_VEL
LIN {X 0,Y 72.576,Z 507.444,A -85,B 0,C 180,E1 -28006.888,E2 -28006.888} C_VEL
LIN {X 0,Y 72.397,Z 507.459,A -85,B 0,C 180,E1 -28012.849,E2 -28012.849} C_VEL
LIN {X 0,Y 72.379,Z 507.463,A -85,B 0,C 180,E1 -28019.082,E2 -28019.082} C_VEL
LIN {X 0,Y 72.302,Z 507.479,A -85,B 0,C 180,E1 -28025.677,E2 -28025.677} C_VEL
LIN {X 0,Y 72.228,Z 507.487,A -85,B 0,C 180,E1 -28032.931,E2 -28032.931} C_VEL
LIN {X 0,Y 72.108,Z 507.501,A -85,B 0,C 180,E1 -28041.236,E2 -28041.236} C_VEL
LIN {X 0,Y 71.955,Z 507.52,A -85,B 0,C 180,E1 -28044.122,E2 -28044.122} C_VEL
LIN {X 0,Y 71.617,Z 507.564,A -85,B 0,C 180,E1 -28052.031,E2 -28052.031} C_VEL
LIN {X 0,Y 73.217,Z 507.459,A -85,B 0,C 180,E1 -28064.027,E2 -28064.027} C_VEL
LIN {X 0,Y 75.967,Z 519.143,A -85,B 0,C 180,E1 -28067.645,E2 -28067.645} C_VEL
LIN {X 0,Y 75.567,Z 527.106,A -85,B 0,C 180,E1 -28071.306,E2 -28071.306} C_VEL
LIN {X 0,Y 75.151,Z 537.889,A -85,B 0,C 180,E1 -28077.319,E2 -28077.319} C_VEL
LIN {X 0,Y 75.339,Z 547.879,A -85,B 0,C 180,E1 -28084.011,E2 -28084.011} C_VEL
LIN {X 0,Y 76.112,Z 556.154,A -85,B 0,C 180,E1 -28090.641,E2 -28090.641} C_VEL
LIN {X 0,Y 77.725,Z 564.405,A -85,B 0,C 180,E1 -28098.449,E2 -28098.449} C_VEL
LIN {X 0,Y 82.361,Z 574.517,A -85,B 0,C 180,E1 -28109.382,E2 -28109.382} C_VEL
LIN {X 0,Y 89.969,Z 582.981,A -85,B 0,C 180,E1 -28118.676,E2 -28118.676} C_VEL
LIN {X 0,Y 95.348,Z 587.13,A -85,B 0,C 180,E1 -28123.078,E2 -28123.078} C_VEL
LIN {X 0,Y 94.395,Z 586.858,A -85,B 0,C 180,E1 -28125.211,E2 -28125.211} C_VEL
LIN {X 0,Y 85.656,Z 581.143,A -85,B 0,C 180,E1 -28134.946,E2 -28134.946} C_VEL
LIN {X 0,Y 81.284,Z 575.529,A -85,B 0,C 180,E1 -28144.385,E2 -28144.385} C_VEL
LIN {X 0,Y 79.749,Z 567.919,A -85,B 0,C 180,E1 -28155.784,E2 -28155.784} C_VEL
LIN {X 0,Y 80.848,Z 560.223,A -85,B 0,C 180,E1 -28165.013,E2 -28165.013} C_VEL
LIN {X 0,Y 82.347,Z 556.432,A -85,B 0,C 180,E1 -28169.236,E2 -28169.236} C_VEL
LIN {X 0,Y 80.372,Z 562.041,A -85,B 0,C 180,E1 -28175.017,E2 -28175.017} C_VEL
LIN {X 0,Y 79.588,Z 568.622,A -85,B 0,C 180,E1 -28182.756,E2 -28182.756} C_VEL
LIN {X 0,Y 80.454,Z 575.595,A -85,B 0,C 180,E1 -28193.147,E2 -28193.147} C_VEL
LIN {X 0,Y 85.567,Z 582.64,A -85,B 0,C 180,E1 -28205.096,E2 -28205.096} C_VEL
LIN {X 0,Y 94.361,Z 588.182,A -85,B 0,C 180,E1 -28214.869,E2 -28214.869} C_VEL
LIN {X 0,Y 95.413,Z 588.507,A -85,B 0,C 180,E1 -28217.007,E2 -28217.007} C_VEL
LIN {X 0,Y 86.324,Z 580.9,A -85,B 0,C 180,E1 -28225.258,E2 -28225.258} C_VEL
LIN {X 0,Y 80.379,Z 572.89,A -85,B 0,C 180,E1 -28234.077,E2 -28234.077} C_VEL
LIN {X 0,Y 77.273,Z 564.825,A -85,B 0,C 180,E1 -28242.808,E2 -28242.808} C_VEL
LIN {X 0,Y 75.776,Z 556.395,A -85,B 0,C 180,E1 -28250.66,E2 -28250.66} C_VEL
LIN {X 0,Y 75.016,Z 546.218,A -85,B 0,C 180,E1 -28258.659,E2 -28258.659} C_VEL
LIN {X 0,Y 75.088,Z 535.65,A -85,B 0,C 180,E1 -28265.372,E2 -28265.372} C_VEL
LIN {X 0,Y 75.878,Z 522.749,A -85,B 0,C 180,E1 -28272.03,E2 -28272.03} C_VEL
LIN {X 0,Y 75.687,Z 519.29,A -85,B 0,C 180,E1 -28273.425,E2 -28273.425} C_VEL
LIN {X 0,Y 72.987,Z 507.391,A -85,B 0,C 180,E1 -28277.153,E2 -28277.153} C_VEL
LIN {X 0,Y 71.604,Z 507.565,A -85,B 0,C 180,E1 -28289.392,E2 -28289.392} C_VEL
LIN {X 0,Y 72.055,Z 507.508,A -85,B 0,C 180,E1 -28298.712,E2 -28298.712} C_VEL
LIN {X 0,Y 72.215,Z 507.489,A -85,B 0,C 180,E1 -28307.059,E2 -28307.059} C_VEL
LIN {X 0,Y 72.302,Z 507.479,A -85,B 0,C 180,E1 -28314.322,E2 -28314.322} C_VEL
LIN {X 0,Y 72.377,Z 507.464,A -85,B 0,C 180,E1 -28320.954,E2 -28320.954} C_VEL
LIN {X 0,Y 72.402,Z 507.458,A -85,B 0,C 180,E1 -28327.153,E2 -28327.153} C_VEL
LIN {X 0,Y 72.76,Z 507.417,A -85,B 0,C 180,E1 -28335.003,E2 -28335.003} C_VEL
LIN {X 0,Y 72.888,Z 507.401,A -85,B 0,C 180,E1 -28338.881,E2 -28338.881} C_VEL
LIN {X 0,Y 72.93,Z 507.385,A -85,B 0,C 180,E1 -28342.807,E2 -28342.807} C_VEL
LIN {X 0,Y 72.354,Z 507.466,A -85,B 0,C 180,E1 -28345.837,E2 -28345.837} C_VEL
LIN {X 0,Y 70.808,Z 507.664,A -85,B 0,C 180,E1 -28348.762,E2 -28348.762} C_VEL
LIN {X 0,Y 66.109,Z 508.248,A -85,B 0,C 180,E1 -28357.068,E2 -28357.068} C_VEL
LIN {X 0,Y 65.735,Z 508.277,A -85,B 0,C 180,E1 -28359.429,E2 -28359.429} C_VEL
LIN {X 0,Y 65.628,Z 508.307,A -85,B 0,C 180,E1 -28365.457,E2 -28365.457} C_VEL
LIN {X 0,Y 65.242,Z 508.358,A -85,B 0,C 180,E1 -28375.524,E2 -28375.524} C_VEL
LIN {X 0,Y 65.2,Z 508.358,A -85,B 0,C 180,E1 -28382.613,E2 -28382.613} C_VEL
LIN {X 0,Y 65.174,Z 508.36,A -85,B 0,C 180,E1 -28390.986,E2 -28390.986} C_VEL
LIN {X 0,Y 65.044,Z 508.375,A -85,B 0,C 180,E1 -28399.584,E2 -28399.584} C_VEL
LIN {X 0,Y 64.583,Z 508.44,A -85,B 0,C 180,E1 -28410.525,E2 -28410.525} C_VEL
LIN {X 0,Y 66.73,Z 508.239,A -85,B 0,C 180,E1 -28426.259,E2 -28426.259} C_VEL
LIN {X 0,Y 69.389,Z 518.934,A -85,B 0,C 180,E1 -28429.789,E2 -28429.789} C_VEL
LIN {X 0,Y 68.899,Z 531.174,A -85,B 0,C 180,E1 -28436.343,E2 -28436.343} C_VEL
LIN {X 0,Y 68.992,Z 541.184,A -85,B 0,C 180,E1 -28442.918,E2 -28442.918} C_VEL
LIN {X 0,Y 69.82,Z 550.359,A -85,B 0,C 180,E1 -28450.144,E2 -28450.144} C_VEL
LIN {X 0,Y 71.481,Z 559.42,A -85,B 0,C 180,E1 -28458.634,E2 -28458.634} C_VEL
LIN {X 0,Y 76.091,Z 570.269,A -85,B 0,C 180,E1 -28470.529,E2 -28470.529} C_VEL
LIN {X 0,Y 84.931,Z 580.265,A -85,B 0,C 180,E1 -28481.451,E2 -28481.451} C_VEL
LIN {X 0,Y 88.005,Z 582.719,A -85,B 0,C 180,E1 -28484.05,E2 -28484.05} C_VEL
LIN {X 0,Y 79.393,Z 576.509,A -85,B 0,C 180,E1 -28494.414,E2 -28494.414} C_VEL
LIN {X 0,Y 75.151,Z 570.158,A -85,B 0,C 180,E1 -28505.113,E2 -28505.113} C_VEL
LIN {X 0,Y 74.182,Z 561.654,A -85,B 0,C 180,E1 -28517.713,E2 -28517.713} C_VEL
LIN {X 0,Y 76.648,Z 552.233,A -85,B 0,C 180,E1 -28528.686,E2 -28528.686} C_VEL
LIN {X 0,Y 76.859,Z 551.935,A -85,B 0,C 180,E1 -28529.181,E2 -28529.181} C_VEL
LIN {X 0,Y 74.892,Z 556.411,A -85,B 0,C 180,E1 -28534.036,E2 -28534.036} C_VEL
LIN {X 0,Y 74.026,Z 562.44,A -85,B 0,C 180,E1 -28540.946,E2 -28540.946} C_VEL
LIN {X 0,Y 74.445,Z 570.217,A -85,B 0,C 180,E1 -28552.186,E2 -28552.186} C_VEL
LIN {X 0,Y 79.115,Z 577.925,A -85,B 0,C 180,E1 -28565.331,E2 -28565.331} C_VEL
LIN {X 0,Y 87.909,Z 584.124,A -85,B 0,C 180,E1 -28576.015,E2 -28576.015} C_VEL
LIN {X 0,Y 81.041,Z 578.011,A -85,B 0,C 180,E1 -28582.625,E2 -28582.625} C_VEL
LIN {X 0,Y 74.684,Z 569.653,A -85,B 0,C 180,E1 -28591.934,E2 -28591.934} C_VEL
LIN {X 0,Y 71.295,Z 561.115,A -85,B 0,C 180,E1 -28601.316,E2 -28601.316} C_VEL
LIN {X 0,Y 69.566,Z 552.247,A -85,B 0,C 180,E1 -28609.818,E2 -28609.818} C_VEL
LIN {X 0,Y 68.759,Z 542.273,A -85,B 0,C 180,E1 -28617.805,E2 -28617.805} C_VEL
LIN {X 0,Y 68.703,Z 531.237,A -85,B 0,C 180,E1 -28625.137,E2 -28625.137} C_VEL
LIN {X 0,Y 69.226,Z 520.257,A -85,B 0,C 180,E1 -28630.975,E2 -28630.975} C_VEL
LIN {X 0,Y 66.334,Z 508.216,A -85,B 0,C 180,E1 -28635.261,E2 -28635.261} C_VEL
LIN {X 0,Y 64.628,Z 508.425,A -85,B 0,C 180,E1 -28652.94,E2 -28652.94} C_VEL
LIN {X 0,Y 64.996,Z 508.38,A -85,B 0,C 180,E1 -28660.807,E2 -28660.807} C_VEL
LIN {X 0,Y 65.189,Z 508.356,A -85,B 0,C 180,E1 -28669.695,E2 -28669.695} C_VEL
LIN {X 0,Y 65.257,Z 508.346,A -85,B 0,C 180,E1 -28679.498,E2 -28679.498} C_VEL
LIN {X 0,Y 65.245,Z 508.357,A -85,B 0,C 180,E1 -28684.477,E2 -28684.477} C_VEL
LIN {X 0,Y 65.654,Z 508.304,A -85,B 0,C 180,E1 -28694.459,E2 -28694.459} C_VEL
LIN {X 0,Y 65.787,Z 508.281,A -85,B 0,C 180,E1 -28697.663,E2 -28697.663} C_VEL
LIN {X 0,Y 66.496,Z 508.203,A -85,B 0,C 180,E1 -28710,E2 -28710} C_VEL
LIN {X 0,Y 65.735,Z 508.277,A -85,B 0,C 180,E1 -28719.429,E2 -28719.429} C_VEL
LIN {X 0,Y 65.348,Z 508.335,A -85,B 0,C 180,E1 -28722.845,E2 -28722.845} C_VEL
LIN {X 0,Y 63.919,Z 508.524,A -85,B 0,C 180,E1 -28727.94,E2 -28727.94} C_VEL
LIN {X 0,Y 61.974,Z 508.768,A -85,B 0,C 180,E1 -28733.079,E2 -28733.079} C_VEL
LIN {X 0,Y 57.969,Z 509.254,A -85,B 0,C 180,E1 -28748.409,E2 -28748.409} C_VEL
LIN {X 0,Y 57.927,Z 509.262,A -85,B 0,C 180,E1 -28756.715,E2 -28756.715} C_VEL
LIN {X 0,Y 57.726,Z 509.295,A -85,B 0,C 180,E1 -28762.499,E2 -28762.499} C_VEL
LIN {X 0,Y 57.527,Z 509.319,A -85,B 0,C 180,E1 -28770.744,E2 -28770.744} C_VEL
LIN {X 0,Y 59.938,Z 509.019,A -85,B 0,C 180,E1 -28788.157,E2 -28788.157} C_VEL
LIN {X 0,Y 60.343,Z 508.97,A -85,B 0,C 180,E1 -28788.983,E2 -28788.983} C_VEL
LIN {X 0,Y 62.588,Z 517.423,A -85,B 0,C 180,E1 -28791.93,E2 -28791.93} C_VEL
LIN {X 0,Y 62.769,Z 520.771,A -85,B 0,C 180,E1 -28793.57,E2 -28793.57} C_VEL
LIN {X 0,Y 62.668,Z 532.376,A -85,B 0,C 180,E1 -28800.802,E2 -28800.802} C_VEL
LIN {X 0,Y 63.252,Z 541.952,A -85,B 0,C 180,E1 -28807.982,E2 -28807.982} C_VEL
LIN {X 0,Y 64.284,Z 549.224,A -85,B 0,C 180,E1 -28814.239,E2 -28814.239} C_VEL
LIN {X 0,Y 66.117,Z 556.751,A -85,B 0,C 180,E1 -28821.84,E2 -28821.84} C_VEL
LIN {X 0,Y 70.761,Z 566.737,A -85,B 0,C 180,E1 -28833.109,E2 -28833.109} C_VEL
LIN {X 0,Y 78.063,Z 575.312,A -85,B 0,C 180,E1 -28842.47,E2 -28842.47} C_VEL
LIN {X 0,Y 80.072,Z 577.142,A -85,B 0,C 180,E1 -28844.6,E2 -28844.6} C_VEL
LIN {X 0,Y 72.923,Z 571.091,A -85,B 0,C 180,E1 -28854.672,E2 -28854.672} C_VEL
LIN {X 0,Y 69.25,Z 564.411,A -85,B 0,C 180,E1 -28866.049,E2 -28866.049} C_VEL
LIN {X 0,Y 68.765,Z 556.149,A -85,B 0,C 180,E1 -28878.205,E2 -28878.205} C_VEL
LIN {X 0,Y 70.405,Z 549.213,A -85,B 0,C 180,E1 -28886.563,E2 -28886.563} C_VEL
LIN {X 0,Y 71.516,Z 547.272,A -85,B 0,C 180,E1 -28889.121,E2 -28889.121} C_VEL
LIN {X 0,Y 69.332,Z 551.807,A -85,B 0,C 180,E1 -28894.359,E2 -28894.359} C_VEL
LIN {X 0,Y 68.361,Z 559.569,A -85,B 0,C 180,E1 -28903.89,E2 -28903.89} C_VEL
LIN {X 0,Y 69.096,Z 566.159,A -85,B 0,C 180,E1 -28914.007,E2 -28914.007} C_VEL
LIN {X 0,Y 72.794,Z 572.732,A -85,B 0,C 180,E1 -28925.4,E2 -28925.4} C_VEL
LIN {X 0,Y 79.486,Z 578.295,A -85,B 0,C 180,E1 -28935.02,E2 -28935.02} C_VEL
LIN {X 0,Y 78.081,Z 576.934,A -85,B 0,C 180,E1 -28937.56,E2 -28937.56} C_VEL
LIN {X 0,Y 69.216,Z 566.128,A -85,B 0,C 180,E1 -28949.491,E2 -28949.491} C_VEL
LIN {X 0,Y 65.924,Z 558.514,A -85,B 0,C 180,E1 -28958.093,E2 -28958.093} C_VEL
LIN {X 0,Y 63.766,Z 549.469,A -85,B 0,C 180,E1 -28967.267,E2 -28967.267} C_VEL
LIN {X 0,Y 62.71,Z 540.143,A -85,B 0,C 180,E1 -28975.18,E2 -28975.18} C_VEL
LIN {X 0,Y 62.389,Z 528.743,A -85,B 0,C 180,E1 -28983.23,E2 -28983.23} C_VEL
LIN {X 0,Y 62.566,Z 519,A -85,B 0,C 180,E1 -28988.887,E2 -28988.887} C_VEL
LIN {X 0,Y 59.973,Z 509.014,A -85,B 0,C 180,E1 -28992.48,E2 -28992.48} C_VEL
LIN {X 0,Y 57.871,Z 509.275,A -85,B 0,C 180,E1 -29001.368,E2 -29001.368} C_VEL
LIN {X 0,Y 57.539,Z 509.311,A -85,B 0,C 180,E1 -29011.24,E2 -29011.24} C_VEL
LIN {X 0,Y 57.685,Z 509.3,A -85,B 0,C 180,E1 -29017.532,E2 -29017.532} C_VEL
LIN {X 0,Y 57.888,Z 509.267,A -85,B 0,C 180,E1 -29023.243,E2 -29023.243} C_VEL
LIN {X 0,Y 57.954,Z 509.266,A -85,B 0,C 180,E1 -29026.689,E2 -29026.689} C_VEL
LIN {X 0,Y 58.025,Z 509.253,A -85,B 0,C 180,E1 -29032.728,E2 -29032.728} C_VEL
LIN {X 0,Y 58.161,Z 509.232,A -85,B 0,C 180,E1 -29037.767,E2 -29037.767} C_VEL
LIN {X 0,Y 58.154,Z 509.235,A -85,B 0,C 180,E1 -29041.092,E2 -29041.092} C_VEL
LIN {X 0,Y 58.54,Z 509.191,A -85,B 0,C 180,E1 -29053.835,E2 -29053.835} C_VEL
LIN {X 0,Y 58.828,Z 509.153,A -85,B 0,C 180,E1 -29063.139,E2 -29063.139} C_VEL
LIN {X 0,Y 59.386,Z 509.088,A -85,B 0,C 180,E1 -29070,E2 -29070} C_VEL
LIN {X 0,Y 58.65,Z 509.162,A -85,B 0,C 180,E1 -29079.154,E2 -29079.154} C_VEL
LIN {X 0,Y 58.519,Z 509.194,A -85,B 0,C 180,E1 -29086.093,E2 -29086.093} C_VEL
LIN {X 0,Y 58.153,Z 509.235,A -85,B 0,C 180,E1 -29098.909,E2 -29098.909} C_VEL
LIN {X 0,Y 58.161,Z 509.232,A -85,B 0,C 180,E1 -29102.233,E2 -29102.233} C_VEL
LIN {X 0,Y 57.969,Z 509.254,A -85,B 0,C 180,E1 -29108.409,E2 -29108.409} C_VEL
LIN {X 0,Y 57.465,Z 509.324,A -85,B 0,C 180,E1 -29112.261,E2 -29112.261} C_VEL
LIN {X 0,Y 55.838,Z 509.528,A -85,B 0,C 180,E1 -29118.009,E2 -29118.009} C_VEL
LIN {X 0,Y 52.453,Z 509.951,A -85,B 0,C 180,E1 -29128.075,E2 -29128.075} C_VEL
LIN {X 0,Y 50.921,Z 510.141,A -85,B 0,C 180,E1 -29139.326,E2 -29139.326} C_VEL
LIN {X 0,Y 51.133,Z 510.099,A -85,B 0,C 180,E1 -29141.611,E2 -29141.611} C_VEL
LIN {X 0,Y 53.727,Z 509.79,A -85,B 0,C 180,E1 -29151.536,E2 -29151.536} C_VEL
LIN {X 0,Y 54.257,Z 509.772,A -85,B 0,C 180,E1 -29152.556,E2 -29152.556} C_VEL
LIN {X 0,Y 56.409,Z 517.335,A -85,B 0,C 180,E1 -29155.356,E2 -29155.356} C_VEL
LIN {X 0,Y 56.625,Z 528.635,A -85,B 0,C 180,E1 -29162.666,E2 -29162.666} C_VEL
LIN {X 0,Y 57.437,Z 538.694,A -85,B 0,C 180,E1 -29170.574,E2 -29170.574} C_VEL
LIN {X 0,Y 59.142,Z 547.417,A -85,B 0,C 180,E1 -29178.666,E2 -29178.666} C_VEL
LIN {X 0,Y 61.61,Z 555.332,A -85,B 0,C 180,E1 -29187.146,E2 -29187.146} C_VEL
LIN {X 0,Y 68.348,Z 566.494,A -85,B 0,C 180,E1 -29199.989,E2 -29199.989} C_VEL
LIN {X 0,Y 72.071,Z 570.53,A -85,B 0,C 180,E1 -29204.353,E2 -29204.353} C_VEL
LIN {X 0,Y 71.524,Z 570.185,A -85,B 0,C 180,E1 -29206.541,E2 -29206.541} C_VEL
LIN {X 0,Y 65.195,Z 562.645,A -85,B 0,C 180,E1 -29219.584,E2 -29219.584} C_VEL
LIN {X 0,Y 63.307,Z 554.96,A -85,B 0,C 180,E1 -29232.224,E2 -29232.224} C_VEL
LIN {X 0,Y 64.712,Z 545.398,A -85,B 0,C 180,E1 -29245.014,E2 -29245.014} C_VEL
LIN {X 0,Y 66.403,Z 542.381,A -85,B 0,C 180,E1 -29248.963,E2 -29248.963} C_VEL
LIN {X 0,Y 63.922,Z 547.189,A -85,B 0,C 180,E1 -29255.03,E2 -29255.03} C_VEL
LIN {X 0,Y 62.925,Z 555.854,A -85,B 0,C 180,E1 -29266.187,E2 -29266.187} C_VEL
LIN {X 0,Y 64.68,Z 563.91,A -85,B 0,C 180,E1 -29279.63,E2 -29279.63} C_VEL
LIN {X 0,Y 69.663,Z 570.287,A -85,B 0,C 180,E1 -29290.978,E2 -29290.978} C_VEL
LIN {X 0,Y 71.403,Z 571.781,A -85,B 0,C 180,E1 -29293.55,E2 -29293.55} C_VEL
LIN {X 0,Y 71.95,Z 572.104,A -85,B 0,C 180,E1 -29295.746,E2 -29295.746} C_VEL
LIN {X 0,Y 64.038,Z 562.299,A -85,B 0,C 180,E1 -29306.721,E2 -29306.721} C_VEL
LIN {X 0,Y 60.317,Z 554.341,A -85,B 0,C 180,E1 -29315.934,E2 -29315.934} C_VEL
LIN {X 0,Y 58.224,Z 546.405,A -85,B 0,C 180,E1 -29324.243,E2 -29324.243} C_VEL
LIN {X 0,Y 56.865,Z 537.98,A -85,B 0,C 180,E1 -29331.92,E2 -29331.92} C_VEL
LIN {X 0,Y 56.224,Z 527.47,A -85,B 0,C 180,E1 -29340.002,E2 -29340.002} C_VEL
LIN {X 0,Y 56.13,Z 518.289,A -85,B 0,C 180,E1 -29345.841,E2 -29345.841} C_VEL
LIN {X 0,Y 53.719,Z 509.793,A -85,B 0,C 180,E1 -29349.177,E2 -29349.177} C_VEL
LIN {X 0,Y 51.41,Z 510.075,A -85,B 0,C 180,E1 -29356.875,E2 -29356.875} C_VEL
LIN {X 0,Y 50.491,Z 510.186,A -85,B 0,C 180,E1 -29373.835,E2 -29373.835} C_VEL
LIN {X 0,Y 50.84,Z 510.146,A -85,B 0,C 180,E1 -29383.727,E2 -29383.727} C_VEL
LIN {X 0,Y 50.906,Z 510.144,A -85,B 0,C 180,E1 -29386.346,E2 -29386.346} C_VEL
LIN {X 0,Y 51.05,Z 510.122,A -85,B 0,C 180,E1 -29396.586,E2 -29396.586} C_VEL
LIN {X 0,Y 51.029,Z 510.124,A -85,B 0,C 180,E1 -29405.595,E2 -29405.595} C_VEL
LIN {X 0,Y 51.485,Z 510.069,A -85,B 0,C 180,E1 -29414.156,E2 -29414.156} C_VEL
LIN {X 0,Y 51.704,Z 510.044,A -85,B 0,C 180,E1 -29422.188,E2 -29422.188} C_VEL
LIN {X 0,Y 52.27,Z 509.975,A -85,B 0,C 180,E1 -29430,E2 -29430} C_VEL
LIN {X 0,Y 51.678,Z 510.047,A -85,B 0,C 180,E1 -29437.816,E2 -29437.816} C_VEL
LIN {X 0,Y 51.389,Z 510.084,A -85,B 0,C 180,E1 -29446.791,E2 -29446.791} C_VEL
LIN {X 0,Y 51.026,Z 510.125,A -85,B 0,C 180,E1 -29454.406,E2 -29454.406} C_VEL
LIN {X 0,Y 51.031,Z 510.128,A -85,B 0,C 180,E1 -29464.273,E2 -29464.273} C_VEL
LIN {X 0,Y 50.931,Z 510.141,A -85,B 0,C 180,E1 -29473.627,E2 -29473.627} C_VEL
LIN {X 0,Y 50.877,Z 510.141,A -85,B 0,C 180,E1 -29476.313,E2 -29476.313} C_VEL
LIN {X 0,Y 50.498,Z 510.185,A -85,B 0,C 180,E1 -29486.62,E2 -29486.62} C_VEL
LIN {X 0,Y 51.133,Z 510.099,A -85,B 0,C 180,E1 -29501.611,E2 -29501.611} C_VEL
LIN {X 0,Y 51.539,Z 510.641,A -85,B 0,C 180,E1 -29505.795,E2 -29505.795} C_VEL
LIN {X 0,Y 51.658,Z 512.572,A -85,B 0,C 180,E1 -29510.702,E2 -29510.702} C_VEL
LIN {X 0,Y 51.524,Z 515.417,A -85,B 0,C 180,E1 -29515.169,E2 -29515.169} C_VEL
LIN {X 0,Y 51.181,Z 519.767,A -85,B 0,C 180,E1 -29520.141,E2 -29520.141} C_VEL
LIN {X 0,Y 51.192,Z 529.763,A -85,B 0,C 180,E1 -29529.114,E2 -29529.114} C_VEL
LIN {X 0,Y 52.712,Z 539.084,A -85,B 0,C 180,E1 -29537.455,E2 -29537.455} C_VEL
LIN {X 0,Y 54.731,Z 546.437,A -85,B 0,C 180,E1 -29544.867,E2 -29544.867} C_VEL
LIN {X 0,Y 58.497,Z 554.991,A -85,B 0,C 180,E1 -29554.796,E2 -29554.796} C_VEL
LIN {X 0,Y 64.86,Z 563.728,A -85,B 0,C 180,E1 -29564.773,E2 -29564.773} C_VEL
LIN {X 0,Y 63.866,Z 562.857,A -85,B 0,C 180,E1 -29568.68,E2 -29568.68} C_VEL
LIN {X 0,Y 59.215,Z 555.572,A -85,B 0,C 180,E1 -29581.657,E2 -29581.657} C_VEL
LIN {X 0,Y 58.114,Z 548.836,A -85,B 0,C 180,E1 -29592.765,E2 -29592.765} C_VEL
LIN {X 0,Y 59.62,Z 540.308,A -85,B 0,C 180,E1 -29604.587,E2 -29604.587} C_VEL
LIN {X 0,Y 61.402,Z 537.318,A -85,B 0,C 180,E1 -29609.003,E2 -29609.003} C_VEL
LIN {X 0,Y 58.959,Z 541.575,A -85,B 0,C 180,E1 -29614.743,E2 -29614.743} C_VEL
LIN {X 0,Y 57.751,Z 551.115,A -85,B 0,C 180,E1 -29627.712,E2 -29627.712} C_VEL
LIN {X 0,Y 59.846,Z 559.586,A -85,B 0,C 180,E1 -29642.298,E2 -29642.298} C_VEL
LIN {X 0,Y 63.698,Z 564.56,A -85,B 0,C 180,E1 -29651.453,E2 -29651.453} C_VEL
LIN {X 0,Y 64.76,Z 565.512,A -85,B 0,C 180,E1 -29655.139,E2 -29655.139} C_VEL
LIN {X 0,Y 57.6,Z 555.552,A -85,B 0,C 180,E1 -29666.699,E2 -29666.699} C_VEL
LIN {X 0,Y 53.852,Z 546.644,A -85,B 0,C 180,E1 -29676.953,E2 -29676.953} C_VEL
LIN {X 0,Y 51.873,Z 538.4,A -85,B 0,C 180,E1 -29685.286,E2 -29685.286} C_VEL
LIN {X 0,Y 50.41,Z 527.155,A -85,B 0,C 180,E1 -29695.003,E2 -29695.003} C_VEL
LIN {X 0,Y 50.043,Z 518.006,A -85,B 0,C 180,E1 -29701.815,E2 -29701.815} C_VEL
LIN {X 0,Y 47.724,Z 510.536,A -85,B 0,C 180,E1 -29704.971,E2 -29704.971} C_VEL
LIN {X 0,Y 46.103,Z 510.739,A -85,B 0,C 180,E1 -29708.771,E2 -29708.771} C_VEL
LIN {X 0,Y 43.357,Z 511.084,A -85,B 0,C 180,E1 -29729.1,E2 -29729.1} C_VEL
LIN {X 0,Y 43.49,Z 511.059,A -85,B 0,C 180,E1 -29740.274,E2 -29740.274} C_VEL
LIN {X 0,Y 43.762,Z 511.024,A -85,B 0,C 180,E1 -29750.029,E2 -29750.029} C_VEL
LIN {X 0,Y 43.826,Z 511.022,A -85,B 0,C 180,E1 -29753.307,E2 -29753.307} C_VEL
LIN {X 0,Y 43.845,Z 511.016,A -85,B 0,C 180,E1 -29761.257,E2 -29761.257} C_VEL
LIN {X 0,Y 44.26,Z 510.972,A -85,B 0,C 180,E1 -29772.321,E2 -29772.321} C_VEL
LIN {X 0,Y 44.555,Z 510.935,A -85,B 0,C 180,E1 -29780.924,E2 -29780.924} C_VEL
LIN {X 0,Y 45.143,Z 510.862,A -85,B 0,C 180,E1 -29790,E2 -29790} C_VEL
LIN {X 0,Y 44.532,Z 510.938,A -85,B 0,C 180,E1 -29799.08,E2 -29799.08} C_VEL
LIN {X 0,Y 44.155,Z 510.983,A -85,B 0,C 180,E1 -29808.562,E2 -29808.562} C_VEL
LIN {X 0,Y 43.844,Z 511.016,A -85,B 0,C 180,E1 -29818.743,E2 -29818.743} C_VEL
LIN {X 0,Y 43.832,Z 511.021,A -85,B 0,C 180,E1 -29826.704,E2 -29826.704} C_VEL
LIN {X 0,Y 43.775,Z 511.022,A -85,B 0,C 180,E1 -29829.955,E2 -29829.955} C_VEL
LIN {X 0,Y 43.536,Z 511.053,A -85,B 0,C 180,E1 -29839.777,E2 -29839.777} C_VEL
LIN {X 0,Y 43.356,Z 511.084,A -85,B 0,C 180,E1 -29850.899,E2 -29850.899} C_VEL
LIN {X 0,Y 45.93,Z 510.761,A -85,B 0,C 180,E1 -29871.196,E2 -29871.196} C_VEL
LIN {X 0,Y 48.467,Z 510.533,A -85,B 0,C 180,E1 -29877.043,E2 -29877.043} C_VEL
LIN {X 0,Y 50.036,Z 515.631,A -85,B 0,C 180,E1 -29878.985,E2 -29878.985} C_VEL
LIN {X 0,Y 50.441,Z 518.901,A -85,B 0,C 180,E1 -29880.861,E2 -29880.861} C_VEL
LIN {X 0,Y 51.192,Z 529.763,A -85,B 0,C 180,E1 -29889.114,E2 -29889.114} C_VEL
LIN {X 0,Y 51.314,Z 534.164,A -85,B 0,C 180,E1 -29893.497,E2 -29893.497} C_VEL
LIN {X 0,Y 51.024,Z 537.928,A -85,B 0,C 180,E1 -29898.645,E2 -29898.645} C_VEL
LIN {X 0,Y 51.998,Z 546.82,A -85,B 0,C 180,E1 -29913.603,E2 -29913.603} C_VEL
LIN {X 0,Y 53.166,Z 549.282,A -85,B 0,C 180,E1 -29916.845,E2 -29916.845} C_VEL
LIN {X 0,Y 58.583,Z 557.069,A -85,B 0,C 180,E1 -29926.036,E2 -29926.036} C_VEL
LIN {X 0,Y 57.759,Z 556.139,A -85,B 0,C 180,E1 -29929.186,E2 -29929.186} C_VEL
LIN {X 0,Y 53.871,Z 548.705,A -85,B 0,C 180,E1 -29942.832,E2 -29942.832} C_VEL
LIN {X 0,Y 53.268,Z 540.505,A -85,B 0,C 180,E1 -29956.095,E2 -29956.095} C_VEL
LIN {X 0,Y 55.573,Z 533.486,A -85,B 0,C 180,E1 -29966.375,E2 -29966.375} C_VEL
LIN {X 0,Y 56.726,Z 531.978,A -85,B 0,C 180,E1 -29968.89,E2 -29968.89} C_VEL
LIN {X 0,Y 53.981,Z 536.302,A -85,B 0,C 180,E1 -29975.182,E2 -29975.182} C_VEL
LIN {X 0,Y 52.629,Z 542.695,A -85,B 0,C 180,E1 -29984.309,E2 -29984.309} C_VEL
LIN {X 0,Y 53.033,Z 548.488,A -85,B 0,C 180,E1 -29993.426,E2 -29993.426} C_VEL
LIN {X 0,Y 55.34,Z 554.958,A -85,B 0,C 180,E1 -30005.298,E2 -30005.298} C_VEL
LIN {X 0,Y 57.928,Z 558.444,A -85,B 0,C 180,E1 -30011.862,E2 -30011.862} C_VEL
LIN {X 0,Y 58.435,Z 558.979,A -85,B 0,C 180,E1 -30013.813,E2 -30013.813} C_VEL
LIN {X 0,Y 52.199,Z 549.905,A -85,B 0,C 180,E1 -30024.564,E2 -30024.564} C_VEL
LIN {X 0,Y 48.587,Z 541.491,A -85,B 0,C 180,E1 -30034.284,E2 -30034.284} C_VEL
LIN {X 0,Y 46.128,Z 532.524,A -85,B 0,C 180,E1 -30043.403,E2 -30043.403} C_VEL
LIN {X 0,Y 44.714,Z 522.828,A -85,B 0,C 180,E1 -30052.097,E2 -30052.097} C_VEL
LIN {X 0,Y 44.302,Z 517.235,A -85,B 0,C 180,E1 -30056.592,E2 -30056.592} C_VEL
LIN {X 0,Y 42.335,Z 511.206,A -85,B 0,C 180,E1 -30059.132,E2 -30059.132} C_VEL
LIN {X 0,Y 38.165,Z 511.731,A -85,B 0,C 180,E1 -30070.614,E2 -30070.614} C_VEL
LIN {X 0,Y 36.332,Z 511.953,A -85,B 0,C 180,E1 -30095.476,E2 -30095.476} C_VEL
LIN {X 0,Y 36.42,Z 511.941,A -85,B 0,C 180,E1 -30099.476,E2 -30099.476} C_VEL
LIN {X 0,Y 36.679,Z 511.905,A -85,B 0,C 180,E1 -30110.04,E2 -30110.04} C_VEL
LIN {X 0,Y 36.713,Z 511.912,A -85,B 0,C 180,E1 -30114.95,E2 -30114.95} C_VEL
LIN {X 0,Y 37.082,Z 511.863,A -85,B 0,C 180,E1 -30131.382,E2 -30131.382} C_VEL
LIN {X 0,Y 37.353,Z 511.825,A -85,B 0,C 180,E1 -30139.155,E2 -30139.155} C_VEL
LIN {X 0,Y 38.002,Z 511.752,A -85,B 0,C 180,E1 -30150,E2 -30150} C_VEL
LIN {X 0,Y 37.329,Z 511.828,A -85,B 0,C 180,E1 -30160.852,E2 -30160.852} C_VEL
LIN {X 0,Y 37.057,Z 511.867,A -85,B 0,C 180,E1 -30168.502,E2 -30168.502} C_VEL
LIN {X 0,Y 36.717,Z 511.912,A -85,B 0,C 180,E1 -30185.046,E2 -30185.046} C_VEL
LIN {X 0,Y 36.691,Z 511.904,A -85,B 0,C 180,E1 -30189.983,E2 -30189.983} C_VEL
LIN {X 0,Y 36.475,Z 511.934,A -85,B 0,C 180,E1 -30200.419,E2 -30200.419} C_VEL
LIN {X 0,Y 36.932,Z 511.879,A -85,B 0,C 180,E1 -30222.078,E2 -30222.078} C_VEL
LIN {X 0,Y 41.509,Z 511.307,A -85,B 0,C 180,E1 -30239.998,E2 -30239.998} C_VEL
LIN {X 0,Y 43.077,Z 511.109,A -85,B 0,C 180,E1 -30242.79,E2 -30242.79} C_VEL
LIN {X 0,Y 44.753,Z 516.341,A -85,B 0,C 180,E1 -30244.989,E2 -30244.989} C_VEL
LIN {X 0,Y 46.003,Z 527.455,A -85,B 0,C 180,E1 -30254.139,E2 -30254.139} C_VEL
LIN {X 0,Y 48.26,Z 537.429,A -85,B 0,C 180,E1 -30263.606,E2 -30263.606} C_VEL
LIN {X 0,Y 50.825,Z 544.474,A -85,B 0,C 180,E1 -30271.228,E2 -30271.228} C_VEL
LIN {X 0,Y 53.166,Z 549.282,A -85,B 0,C 180,E1 -30276.845,E2 -30276.845} C_VEL
LIN {X 0,Y 53.63,Z 550.44,A -85,B 0,C 180,E1 -30279.2,E2 -30279.2} C_VEL
LIN {X 0,Y 53.45,Z 550.803,A -85,B 0,C 180,E1 -30282.922,E2 -30282.922} C_VEL
LIN {X 0,Y 52.565,Z 549.9,A -85,B 0,C 180,E1 -30287.894,E2 -30287.894} C_VEL
LIN {X 0,Y 51.638,Z 548.43,A -85,B 0,C 180,E1 -30291.726,E2 -30291.726} C_VEL
LIN {X 0,Y 49.38,Z 543.521,A -85,B 0,C 180,E1 -30300.759,E2 -30300.759} C_VEL
LIN {X 0,Y 48.399,Z 538.001,A -85,B 0,C 180,E1 -30309.964,E2 -30309.964} C_VEL
LIN {X 0,Y 49.671,Z 530.419,A -85,B 0,C 180,E1 -30322.06,E2 -30322.06} C_VEL
LIN {X 0,Y 52.246,Z 526.503,A -85,B 0,C 180,E1 -30328.808,E2 -30328.808} C_VEL
LIN {X 0,Y 49.396,Z 530.539,A -85,B 0,C 180,E1 -30335.172,E2 -30335.172} C_VEL
LIN {X 0,Y 47.763,Z 536.845,A -85,B 0,C 180,E1 -30345.168,E2 -30345.168} C_VEL
LIN {X 0,Y 48.349,Z 543.457,A -85,B 0,C 180,E1 -30355.854,E2 -30355.854} C_VEL
LIN {X 0,Y 51.634,Z 550.857,A -85,B 0,C 180,E1 -30370.144,E2 -30370.144} C_VEL
LIN {X 0,Y 52.405,Z 551.875,A -85,B 0,C 180,E1 -30372.11,E2 -30372.11} C_VEL
LIN {X 0,Y 49.527,Z 548.006,A -85,B 0,C 180,E1 -30376.998,E2 -30376.998} C_VEL
LIN {X 0,Y 44.999,Z 539.607,A -85,B 0,C 180,E1 -30386.866,E2 -30386.866} C_VEL
LIN {X 0,Y 41.783,Z 530.653,A -85,B 0,C 180,E1 -30396.48,E2 -30396.48} C_VEL
LIN {X 0,Y 39.596,Z 520.948,A -85,B 0,C 180,E1 -30405.877,E2 -30405.877} C_VEL
LIN {X 0,Y 39.055,Z 516.723,A -85,B 0,C 180,E1 -30409.635,E2 -30409.635} C_VEL
LIN {X 0,Y 37.38,Z 511.825,A -85,B 0,C 180,E1 -30411.863,E2 -30411.863} C_VEL
LIN {X 0,Y 33.577,Z 512.287,A -85,B 0,C 180,E1 -30420.003,E2 -30420.003} C_VEL
LIN {X 0,Y 29.139,Z 512.706,A -85,B 0,C 180,E1 -30448.844,E2 -30448.844} C_VEL
LIN {X 0,Y 29.363,Z 512.686,A -85,B 0,C 180,E1 -30465.898,E2 -30465.898} C_VEL
LIN {X 0,Y 29.505,Z 512.671,A -85,B 0,C 180,E1 -30481.549,E2 -30481.549} C_VEL
LIN {X 0,Y 29.891,Z 512.635,A -85,B 0,C 180,E1 -30490.141,E2 -30490.141} C_VEL
LIN {X 0,Y 30.13,Z 512.611,A -85,B 0,C 180,E1 -30496.511,E2 -30496.511} C_VEL
LIN {X 0,Y 30.819,Z 512.551,A -85,B 0,C 180,E1 -30510,E2 -30510} C_VEL
LIN {X 0,Y 30.107,Z 512.614,A -85,B 0,C 180,E1 -30523.499,E2 -30523.499} C_VEL
LIN {X 0,Y 29.865,Z 512.638,A -85,B 0,C 180,E1 -30529.72,E2 -30529.72} C_VEL
LIN {X 0,Y 29.493,Z 512.672,A -85,B 0,C 180,E1 -30538.463,E2 -30538.463} C_VEL
LIN {X 0,Y 29.36,Z 512.685,A -85,B 0,C 180,E1 -30555.9,E2 -30555.9} C_VEL
LIN {X 0,Y 29.138,Z 512.707,A -85,B 0,C 180,E1 -30571.154,E2 -30571.154} C_VEL
LIN {X 0,Y 35.274,Z 512.085,A -85,B 0,C 180,E1 -30605.001,E2 -30605.001} C_VEL
LIN {X 0,Y 38.379,Z 511.703,A -85,B 0,C 180,E1 -30610.216,E2 -30610.216} C_VEL
LIN {X 0,Y 39.578,Z 515.104,A -85,B 0,C 180,E1 -30611.521,E2 -30611.521} C_VEL
LIN {X 0,Y 41.2,Z 524.601,A -85,B 0,C 180,E1 -30619.945,E2 -30619.945} C_VEL
LIN {X 0,Y 44.372,Z 535.017,A -85,B 0,C 180,E1 -30630.33,E2 -30630.33} C_VEL
LIN {X 0,Y 47.751,Z 542.503,A -85,B 0,C 180,E1 -30638.657,E2 -30638.657} C_VEL
LIN {X 0,Y 51.683,Z 548.671,A -85,B 0,C 180,E1 -30646.011,E2 -30646.011} C_VEL
LIN {X 0,Y 52.667,Z 549.984,A -85,B 0,C 180,E1 -30648.148,E2 -30648.148} C_VEL
LIN {X 0,Y 49.03,Z 542.531,A -85,B 0,C 180,E1 -30662.232,E2 -30662.232} C_VEL
LIN {X 0,Y 48.399,Z 538.001,A -85,B 0,C 180,E1 -30669.964,E2 -30669.964} C_VEL
LIN {X 0,Y 47.959,Z 535.229,A -85,B 0,C 180,E1 -30673.448,E2 -30673.448} C_VEL
LIN {X 0,Y 46.083,Z 525.089,A -85,B 0,C 180,E1 -30682.247,E2 -30682.247} C_VEL
LIN {X 0,Y 46.639,Z 522.56,A -85,B 0,C 180,E1 -30685.359,E2 -30685.359} C_VEL
LIN {X 0,Y 47.116,Z 521.83,A -85,B 0,C 180,E1 -30686.559,E2 -30686.559} C_VEL
LIN {X 0,Y 48.069,Z 520.746,A -85,B 0,C 180,E1 -30688.56,E2 -30688.56} C_VEL
LIN {X 0,Y 44.966,Z 524.8,A -85,B 0,C 180,E1 -30695.683,E2 -30695.683} C_VEL
LIN {X 0,Y 43.145,Z 530.952,A -85,B 0,C 180,E1 -30706.466,E2 -30706.466} C_VEL
LIN {X 0,Y 43.93,Z 538.139,A -85,B 0,C 180,E1 -30718.682,E2 -30718.682} C_VEL
LIN {X 0,Y 45.805,Z 542.775,A -85,B 0,C 180,E1 -30727.86,E2 -30727.86} C_VEL
LIN {X 0,Y 46.518,Z 544.026,A -85,B 0,C 180,E1 -30730.941,E2 -30730.941} C_VEL
LIN {X 0,Y 41.359,Z 535.788,A -85,B 0,C 180,E1 -30740.418,E2 -30740.418} C_VEL
LIN {X 0,Y 37.814,Z 527.42,A -85,B 0,C 180,E1 -30749.265,E2 -30749.265} C_VEL
LIN {X 0,Y 34.918,Z 517.288,A -85,B 0,C 180,E1 -30759.379,E2 -30759.379} C_VEL
LIN {X 0,Y 34.124,Z 514.307,A -85,B 0,C 180,E1 -30761.721,E2 -30761.721} C_VEL
LIN {X 0,Y 33.248,Z 512.319,A -85,B 0,C 180,E1 -30762.512,E2 -30762.512} C_VEL
LIN {X 0,Y 28.488,Z 512.767,A -85,B 0,C 180,E1 -30770.678,E2 -30770.678} C_VEL
LIN {X 0,Y 22.401,Z 513.078,A -85,B 0,C 180,E1 -30799.746,E2 -30799.746} C_VEL
LIN {X 0,Y 21.954,Z 513.092,A -85,B 0,C 180,E1 -30819.817,E2 -30819.817} C_VEL
LIN {X 0,Y 22.084,Z 513.088,A -85,B 0,C 180,E1 -30830.471,E2 -30830.471} C_VEL
LIN {X 0,Y 22.844,Z 513.064,A -85,B 0,C 180,E1 -30852.082,E2 -30852.082} C_VEL
LIN {X 0,Y 23.588,Z 513.042,A -85,B 0,C 180,E1 -30870,E2 -30870} C_VEL
LIN {X 0,Y 22.813,Z 513.065,A -85,B 0,C 180,E1 -30887.943,E2 -30887.943} C_VEL
LIN {X 0,Y 22.097,Z 513.088,A -85,B 0,C 180,E1 -30909.502,E2 -30909.502} C_VEL
LIN {X 0,Y 21.971,Z 513.092,A -85,B 0,C 180,E1 -30920.221,E2 -30920.221} C_VEL
LIN {X 0,Y 22.512,Z 513.074,A -85,B 0,C 180,E1 -30941.804,E2 -30941.804} C_VEL
LIN {X 0,Y 30.11,Z 512.615,A -85,B 0,C 180,E1 -30973.495,E2 -30973.495} C_VEL
LIN {X 0,Y 34.493,Z 512.178,A -85,B 0,C 180,E1 -30979.526,E2 -30979.526} C_VEL
LIN {X 0,Y 35.301,Z 514.235,A -85,B 0,C 180,E1 -30980.387,E2 -30980.387} C_VEL
LIN {X 0,Y 38.182,Z 524.824,A -85,B 0,C 180,E1 -30990.407,E2 -30990.407} C_VEL
LIN {X 0,Y 41.71,Z 533.456,A -85,B 0,C 180,E1 -30999.185,E2 -30999.185} C_VEL
LIN {X 0,Y 45.99,Z 540.795,A -85,B 0,C 180,E1 -31007.399,E2 -31007.399} C_VEL
LIN {X 0,Y 46.774,Z 541.91,A -85,B 0,C 180,E1 -31008.698,E2 -31008.698} C_VEL
LIN {X 0,Y 46.144,Z 540.702,A -85,B 0,C 180,E1 -31012.467,E2 -31012.467} C_VEL
LIN {X 0,Y 44.008,Z 533.647,A -85,B 0,C 180,E1 -31025.663,E2 -31025.663} C_VEL
LIN {X 0,Y 44.589,Z 526.357,A -85,B 0,C 180,E1 -31038.407,E2 -31038.407} C_VEL
LIN {X 0,Y 47.116,Z 521.83,A -85,B 0,C 180,E1 -31046.559,E2 -31046.559} C_VEL
LIN {X 0,Y 47.007,Z 521.093,A -85,B 0,C 180,E1 -31048.549,E2 -31048.549} C_VEL
LIN {X 0,Y 45.33,Z 520.738,A -85,B 0,C 180,E1 -31051.481,E2 -31051.481} C_VEL
LIN {X 0,Y 42.147,Z 521.434,A -85,B 0,C 180,E1 -31056.655,E2 -31056.655} C_VEL
LIN {X 0,Y 39.896,Z 523.016,A -85,B 0,C 180,E1 -31062.168,E2 -31062.168} C_VEL
LIN {X 0,Y 38.813,Z 525.208,A -85,B 0,C 180,E1 -31068.198,E2 -31068.198} C_VEL
LIN {X 0,Y 38.701,Z 527.057,A -85,B 0,C 180,E1 -31072.062,E2 -31072.062} C_VEL
LIN {X 0,Y 40.81,Z 535.063,A -85,B 0,C 180,E1 -31087.073,E2 -31087.073} C_VEL
LIN {X 0,Y 40.241,Z 534.415,A -85,B 0,C 180,E1 -31090.011,E2 -31090.011} C_VEL
LIN {X 0,Y 35.696,Z 526.417,A -85,B 0,C 180,E1 -31098.361,E2 -31098.361} C_VEL
LIN {X 0,Y 31.754,Z 516.298,A -85,B 0,C 180,E1 -31108.292,E2 -31108.292} C_VEL
LIN {X 0,Y 31.101,Z 514.144,A -85,B 0,C 180,E1 -31110.379,E2 -31110.379} C_VEL
LIN {X 0,Y 30.241,Z 512.601,A -85,B 0,C 180,E1 -31110.887,E2 -31110.887} C_VEL
LIN {X 0,Y 22.109,Z 513.087,A -85,B 0,C 180,E1 -31122.487,E2 -31122.487} C_VEL
LIN {X 0,Y 14.773,Z 513.178,A -85,B 0,C 180,E1 -31168.415,E2 -31168.415} C_VEL
LIN {X 0,Y 15.035,Z 513.178,A -85,B 0,C 180,E1 -31202.132,E2 -31202.132} C_VEL
LIN {X 0,Y 15.256,Z 513.178,A -85,B 0,C 180,E1 -31207.14,E2 -31207.14} C_VEL
LIN {X 0,Y 16.257,Z 513.178,A -85,B 0,C 180,E1 -31230,E2 -31230} C_VEL
LIN {X 0,Y 15.246,Z 513.178,A -85,B 0,C 180,E1 -31252.767,E2 -31252.767} C_VEL
LIN {X 0,Y 15.028,Z 513.178,A -85,B 0,C 180,E1 -31257.883,E2 -31257.883} C_VEL
LIN {X 0,Y 14.775,Z 513.178,A -85,B 0,C 180,E1 -31291.59,E2 -31291.59} C_VEL
LIN {X 0,Y 22.243,Z 513.083,A -85,B 0,C 180,E1 -31338.415,E2 -31338.415} C_VEL
LIN {X 0,Y 31.155,Z 512.516,A -85,B 0,C 180,E1 -31350.498,E2 -31350.498} C_VEL
LIN {X 0,Y 31.782,Z 512.457,A -85,B 0,C 180,E1 -31350.867,E2 -31350.867} C_VEL
LIN {X 0,Y 33.982,Z 518.73,A -85,B 0,C 180,E1 -31356.481,E2 -31356.481} C_VEL
LIN {X 0,Y 37.655,Z 527.018,A -85,B 0,C 180,E1 -31364.416,E2 -31364.416} C_VEL
LIN {X 0,Y 40.867,Z 532.586,A -85,B 0,C 180,E1 -31369.941,E2 -31369.941} C_VEL
LIN {X 0,Y 41.527,Z 533.471,A -85,B 0,C 180,E1 -31372.153,E2 -31372.153} C_VEL
LIN {X 0,Y 39.614,Z 524.492,A -85,B 0,C 180,E1 -31389.217,E2 -31389.217} C_VEL
LIN {X 0,Y 41.604,Z 517.842,A -85,B 0,C 180,E1 -31402.364,E2 -31402.364} C_VEL
LIN {X 0,Y 43.991,Z 514.964,A -85,B 0,C 180,E1 -31408.549,E2 -31408.549} C_VEL
LIN {X 0,Y 40.709,Z 518.963,A -85,B 0,C 180,E1 -31416.534,E2 -31416.534} C_VEL
LIN {X 0,Y 38.701,Z 527.057,A -85,B 0,C 180,E1 -31432.062,E2 -31432.062} C_VEL
LIN {X 0,Y 38.361,Z 527.693,A -85,B 0,C 180,E1 -31434.729,E2 -31434.729} C_VEL
LIN {X 0,Y 37.366,Z 527.271,A -85,B 0,C 180,E1 -31438.381,E2 -31438.381} C_VEL
LIN {X 0,Y 35.626,Z 525.352,A -85,B 0,C 180,E1 -31443.136,E2 -31443.136} C_VEL
LIN {X 0,Y 33.551,Z 522.119,A -85,B 0,C 180,E1 -31447.672,E2 -31447.672} C_VEL
LIN {X 0,Y 30.838,Z 516.89,A -85,B 0,C 180,E1 -31453.6,E2 -31453.6} C_VEL
LIN {X 0,Y 29.607,Z 514.079,A -85,B 0,C 180,E1 -31456.33,E2 -31456.33} C_VEL
LIN {X 0,Y 28.986,Z 512.721,A -85,B 0,C 180,E1 -31457.34,E2 -31457.34} C_VEL
LIN {X 0,Y 16.515,Z 513.178,A -85,B 0,C 180,E1 -31468.331,E2 -31468.331} C_VEL
LIN {X 0,Y 7.651,Z 513.178,A -85,B 0,C 180,E1 -31523.289,E2 -31523.289} C_VEL
LIN {X 0,Y 7.729,Z 513.178,A -85,B 0,C 180,E1 -31565.436,E2 -31565.436} C_VEL
LIN {X 0,Y 8.681,Z 513.178,A -85,B 0,C 180,E1 -31590,E2 -31590} C_VEL
LIN {X 0,Y 7.727,Z 513.178,A -85,B 0,C 180,E1 -31614.529,E2 -31614.529} C_VEL
LIN {X 0,Y 7.652,Z 513.178,A -85,B 0,C 180,E1 -31656.701,E2 -31656.701} C_VEL
LIN {X 0,Y 22.158,Z 513.086,A -85,B 0,C 180,E1 -31719.367,E2 -31719.367} C_VEL
LIN {X 0,Y 30.694,Z 512.624,A -85,B 0,C 180,E1 -31724.521,E2 -31724.521} C_VEL
LIN {X 0,Y 35.368,Z 522.273,A -85,B 0,C 180,E1 -31732.637,E2 -31732.637} C_VEL
LIN {X 0,Y 36.572,Z 524.24,A -85,B 0,C 180,E1 -31734.795,E2 -31734.795} C_VEL
LIN {X 0,Y 35.804,Z 516.888,A -85,B 0,C 180,E1 -31750.051,E2 -31750.051} C_VEL
LIN {X 0,Y 37.738,Z 511.775,A -85,B 0,C 180,E1 -31761.576,E2 -31761.576} C_VEL
LIN {X 0,Y 37.074,Z 511.861,A -85,B 0,C 180,E1 -31772.505,E2 -31772.505} C_VEL
LIN {X 0,Y 37.398,Z 511.892,A -85,B 0,C 180,E1 -31775.21,E2 -31775.21} C_VEL
LIN {X 0,Y 34.846,Z 518.064,A -85,B 0,C 180,E1 -31788.512,E2 -31788.512} C_VEL
LIN {X 0,Y 35.122,Z 523.728,A -85,B 0,C 180,E1 -31800.536,E2 -31800.536} C_VEL
LIN {X 0,Y 35.079,Z 524.964,A -85,B 0,C 180,E1 -31806.74,E2 -31806.74} C_VEL
LIN {X 0,Y 29.607,Z 514.079,A -85,B 0,C 180,E1 -31816.33,E2 -31816.33} C_VEL
LIN {X 0,Y 28.281,Z 513.151,A -85,B 0,C 180,E1 -31817.261,E2 -31817.261} C_VEL
LIN {X 0,Y 25.818,Z 512.972,A -85,B 0,C 180,E1 -31817.366,E2 -31817.366} C_VEL
LIN {X 0,Y 13.143,Z 513.296,A -85,B 0,C 180,E1 -31807.201,E2 -31807.201} C_VEL
LIN {X 0,Y 9.336,Z 513.183,A -85,B 0,C 180,E1 -31804.619,E2 -31804.619} C_VEL
LIN {X 0,Y 8.568,Z 513.178,A -85,B 0,C 180,E1 -31804.802,E2 -31804.802} C_VEL
LIN {X 0,Y 0.13,Z 513.178,A -85,B 0,C 180,E1 -31950,E2 -31950} C_VEL
LIN {X 0,Y 8.517,Z 513.178,A -85,B 0,C 180,E1 -32095.586,E2 -32095.586} C_VEL
LIN {X 0,Y 24.918,Z 513,A -85,B 0,C 180,E1 -32097.787,E2 -32097.787} C_VEL
LIN {X 0,Y 31.371,Z 512.499,A -85,B 0,C 180,E1 -32098.562,E2 -32098.562} C_VEL
LIN {X 0,Y 31.758,Z 513.212,A -85,B 0,C 180,E1 -32099.036,E2 -32099.036} C_VEL
LIN {X 0,Y 32.057,Z 513.183,A -85,B 0,C 180,E1 -32101.268,E2 -32101.268} C_VEL
LIN {X 0,Y 31.952,Z 512.439,A -85,B 0,C 180,E1 -32103.224,E2 -32103.224} C_VEL
LIN {X 0,Y 30.94,Z 512.536,A -85,B 0,C 180,E1 -32105.305,E2 -32105.305} C_VEL
LIN {X 0,Y 29.688,Z 512.654,A -85,B 0,C 180,E1 -32111.237,E2 -32111.237} C_VEL
LIN {X 0,Y 30.089,Z 512.615,A -85,B 0,C 180,E1 -32130,E2 -32130} C_VEL
LIN {X 0,Y 29.082,Z 512.711,A -85,B 0,C 180,E1 -32144.849,E2 -32144.849} C_VEL
LIN {X 0,Y 30.496,Z 512.581,A -85,B 0,C 180,E1 -32151.82,E2 -32151.82} C_VEL
LIN {X 0,Y 31.036,Z 512.616,A -85,B 0,C 180,E1 -32153.098,E2 -32153.098} C_VEL
LIN {X 0,Y 31.02,Z 514.174,A -85,B 0,C 180,E1 -32156.944,E2 -32156.944} C_VEL
LIN {X 0,Y 30.836,Z 515.077,A -85,B 0,C 180,E1 -32160.93,E2 -32160.93} C_VEL
LIN {X 0,Y 29.455,Z 512.676,A -85,B 0,C 180,E1 -32162.592,E2 -32162.592} C_VEL
LIN {X 0,Y 25.129,Z 512.993,A -85,B 0,C 180,E1 -32162.969,E2 -32162.969} C_VEL
LIN {X 0,Y 8.568,Z 513.178,A -85,B 0,C 180,E1 -32164.802,E2 -32164.802} C_VEL
LIN {X 0,Y 7.649,Z 513.18,A -85,B 0,C 180,E1 -32158.171,E2 -32158.171} C_VEL
LIN {X 0,Y 8.263,Z 513.184,A -85,B 0,C 180,E1 -32140.299,E2 -32140.299} C_VEL
LIN {X 0,Y 14.215,Z 513.178,A -85,B 0,C 180,E1 -32121.063,E2 -32121.063} C_VEL
LIN {X 0,Y 21.34,Z 513.118,A -85,B 0,C 180,E1 -32116.581,E2 -32116.581} C_VEL
LIN {X 0,Y 21.649,Z 513.101,A -85,B 0,C 180,E1 -32116.864,E2 -32116.864} C_VEL
LIN {X 0,Y 12.904,Z 513.178,A -85,B 0,C 180,E1 -32130,E2 -32130} C_VEL
LIN {X 0,Y 21.718,Z 513.098,A -85,B 0,C 180,E1 -32143.892,E2 -32143.892} C_VEL
